LIN {X 0,Y 466.737,Z 357.71,A -85,B 0,C 180,E1 -7511.495,E2 -7511.495} C_VEL
LIN {X 0,Y 466.868,Z 355.189,A -85,B 0,C 180,E1 -7512.642,E2 -7512.642} C_VEL
LIN {X 0,Y 467.016,Z 350.85,A -85,B 0,C 180,E1 -7514.108,E2 -7514.108} C_VEL
LIN {X 0,Y 467.238,Z 344.895,A -85,B 0,C 180,E1 -7515.6,E2 -7515.6} C_VEL
LIN {X 0,Y 467.572,Z 338.558,A -85,B 0,C 180,E1 -7516.852,E2 -7516.852} C_VEL
LIN {X 0,Y 468.005,Z 329.992,A -85,B 0,C 180,E1 -7518.213,E2 -7518.213} C_VEL
LIN {X 0,Y 468.461,Z 320.576,A -85,B 0,C 180,E1 -7519.404,E2 -7519.404} C_VEL
LIN {X 0,Y 468.938,Z 310.487,A -85,B 0,C 180,E1 -7520.436,E2 -7520.436} C_VEL
LIN {X 0,Y 469.406,Z 299.87,A -85,B 0,C 180,E1 -7521.312,E2 -7521.312} C_VEL
LIN {X 0,Y 469.889,Z 288.638,A -85,B 0,C 180,E1 -7522.042,E2 -7522.042} C_VEL
LIN {X 0,Y 470.257,Z 275.513,A -85,B 0,C 180,E1 -7522.685,E2 -7522.685} C_VEL
LIN {X 0,Y 470.519,Z 262.558,A -85,B 0,C 180,E1 -7523.128,E2 -7523.128} C_VEL
LIN {X 0,Y 470.697,Z 246.728,A -85,B 0,C 180,E1 -7523.438,E2 -7523.438} C_VEL
LIN {X 0,Y 471.435,Z 164.016,A -85,B 0,C 180,E1 -7524.746,E2 -7524.746} C_VEL
LIN {X 0,Y 468.633,Z 150.697,A -85,B 0,C 180,E1 -7525.095,E2 -7525.095} C_VEL
LIN {X 0,Y 468.758,Z 142.318,A -85,B 0,C 180,E1 -7526.795,E2 -7526.795} C_VEL
LIN {X 0,Y 467.609,Z 135.273,A -85,B 0,C 180,E1 -7528.289,E2 -7528.289} C_VEL
LIN {X 0,Y 467.577,Z 135.244,A -85,B 0,C 180,E1 -7531.251,E2 -7531.251} C_VEL
LIN {X 0,Y 467.591,Z 135.241,A -85,B 0,C 180,E1 -7534.159,E2 -7534.159} C_VEL
LIN {X 0,Y 467.579,Z 135.247,A -85,B 0,C 180,E1 -7536.997,E2 -7536.997} C_VEL
LIN {X 0,Y 467.625,Z 135.234,A -85,B 0,C 180,E1 -7539.778,E2 -7539.778} C_VEL
LIN {X 0,Y 467.598,Z 135.239,A -85,B 0,C 180,E1 -7542.507,E2 -7542.507} C_VEL
LIN {X 0,Y 467.606,Z 135.24,A -85,B 0,C 180,E1 -7545.197,E2 -7545.197} C_VEL
LIN {X 0,Y 467.66,Z 135.231,A -85,B 0,C 180,E1 -7547.855,E2 -7547.855} C_VEL
LIN {X 0,Y 467.671,Z 135.229,A -85,B 0,C 180,E1 -7551.358,E2 -7551.358} C_VEL
LIN {X 0,Y 467.709,Z 135.225,A -85,B 0,C 180,E1 -7553.963,E2 -7553.963} C_VEL
LIN {X 0,Y 467.818,Z 135.209,A -85,B 0,C 180,E1 -7557.417,E2 -7557.417} C_VEL
LIN {X 0,Y 467.854,Z 135.204,A -85,B 0,C 180,E1 -7560,E2 -7560} C_VEL
LIN {X 0,Y 467.816,Z 135.207,A -85,B 0,C 180,E1 -7562.584,E2 -7562.584} C_VEL
LIN {X 0,Y 467.705,Z 135.225,A -85,B 0,C 180,E1 -7566.038,E2 -7566.038} C_VEL
LIN {X 0,Y 467.634,Z 135.231,A -85,B 0,C 180,E1 -7568.644,E2 -7568.644} C_VEL
LIN {X 0,Y 467.646,Z 135.232,A -85,B 0,C 180,E1 -7572.146,E2 -7572.146} C_VEL
LIN {X 0,Y 467.581,Z 135.239,A -85,B 0,C 180,E1 -7575.697,E2 -7575.697} C_VEL
LIN {X 0,Y 467.553,Z 135.239,A -85,B 0,C 180,E1 -7578.739,E2 -7578.739} C_VEL
LIN {X 0,Y 467.52,Z 135.246,A -85,B 0,C 180,E1 -7582.075,E2 -7582.075} C_VEL
LIN {X 0,Y 467.533,Z 135.244,A -85,B 0,C 180,E1 -7584.892,E2 -7584.892} C_VEL
LIN {X 0,Y 467.542,Z 135.241,A -85,B 0,C 180,E1 -7587.775,E2 -7587.775} C_VEL
LIN {X 0,Y 467.534,Z 135.247,A -85,B 0,C 180,E1 -7591.037,E2 -7591.037} C_VEL
LIN {X 0,Y 467.571,Z 135.239,A -85,B 0,C 180,E1 -7593.79,E2 -7593.79} C_VEL
LIN {X 0,Y 467.529,Z 135.25,A -85,B 0,C 180,E1 -7596.963,E2 -7596.963} C_VEL
LIN {X 0,Y 467.568,Z 135.24,A -85,B 0,C 180,E1 -7599.951,E2 -7599.951} C_VEL
LIN {X 0,Y 467.524,Z 135.251,A -85,B 0,C 180,E1 -7602.568,E2 -7602.568} C_VEL
LIN {X 0,Y 467.57,Z 135.244,A -85,B 0,C 180,E1 -7605.052,E2 -7605.052} C_VEL
LIN {X 0,Y 467.571,Z 135.245,A -85,B 0,C 180,E1 -7608.725,E2 -7608.725} C_VEL
LIN {X 0,Y 467.566,Z 135.244,A -85,B 0,C 180,E1 -7611.955,E2 -7611.955} C_VEL
LIN {X 0,Y 467.567,Z 135.241,A -85,B 0,C 180,E1 -7615.167,E2 -7615.167} C_VEL
LIN {X 0,Y 467.587,Z 135.247,A -85,B 0,C 180,E1 -7618.26,E2 -7618.26} C_VEL
LIN {X 0,Y 467.56,Z 135.243,A -85,B 0,C 180,E1 -7621.249,E2 -7621.249} C_VEL
LIN {X 0,Y 467.611,Z 135.331,A -85,B 0,C 180,E1 -7623.65,E2 -7623.65} C_VEL
LIN {X 0,Y 469.706,Z 145.922,A -85,B 0,C 180,E1 -7625.6,E2 -7625.6} C_VEL
LIN {X 0,Y 469.617,Z 153.321,A -85,B 0,C 180,E1 -7626.868,E2 -7626.868} C_VEL
LIN {X 0,Y 468.886,Z 169.647,A -85,B 0,C 180,E1 -7629.605,E2 -7629.605} C_VEL
LIN {X 0,Y 468.398,Z 184.571,A -85,B 0,C 180,E1 -7632.085,E2 -7632.085} C_VEL
LIN {X 0,Y 468.222,Z 189.663,A -85,B 0,C 180,E1 -7632.927,E2 -7632.927} C_VEL
LIN {X 0,Y 471.192,Z 210.245,A -85,B 0,C 180,E1 -7633.383,E2 -7633.383} C_VEL
LIN {X 0,Y 470.478,Z 298.444,A -85,B 0,C 180,E1 -7634.79,E2 -7634.79} C_VEL
LIN {X 0,Y 470.078,Z 311.692,A -85,B 0,C 180,E1 -7635.165,E2 -7635.165} C_VEL
LIN {X 0,Y 469.572,Z 324.447,A -85,B 0,C 180,E1 -7635.702,E2 -7635.702} C_VEL
LIN {X 0,Y 469.102,Z 335.815,A -85,B 0,C 180,E1 -7636.351,E2 -7636.351} C_VEL
LIN {X 0,Y 468.602,Z 347.595,A -85,B 0,C 180,E1 -7637.222,E2 -7637.222} C_VEL
LIN {X 0,Y 468.114,Z 358.121,A -85,B 0,C 180,E1 -7638.196,E2 -7638.196} C_VEL
LIN {X 0,Y 467.705,Z 366.768,A -85,B 0,C 180,E1 -7639.173,E2 -7639.173} C_VEL
LIN {X 0,Y 467.358,Z 374.752,A -85,B 0,C 180,E1 -7640.26,E2 -7640.26} C_VEL
LIN {X 0,Y 467.021,Z 382.558,A -85,B 0,C 180,E1 -7641.562,E2 -7641.562} C_VEL
LIN {X 0,Y 466.83,Z 389.753,A -85,B 0,C 180,E1 -7643.082,E2 -7643.082} C_VEL
LIN {X 0,Y 466.724,Z 394.545,A -85,B 0,C 180,E1 -7644.383,E2 -7644.383} C_VEL
LIN {X 0,Y 466.648,Z 398.21,A -85,B 0,C 180,E1 -7645.681,E2 -7645.681} C_VEL
LIN {X 0,Y 466.701,Z 400.106,A -85,B 0,C 180,E1 -7646.546,E2 -7646.546} C_VEL
LIN {X 0,Y 466.685,Z 401.527,A -85,B 0,C 180,E1 -7647.41,E2 -7647.41} C_VEL
LIN {X 0,Y 466.663,Z 402.544,A -85,B 0,C 180,E1 -7648.273,E2 -7648.273} C_VEL
LIN {X 0,Y 466.627,Z 403.166,A -85,B 0,C 180,E1 -7649.137,E2 -7649.137} C_VEL
LIN {X 0,Y 466.611,Z 403.39,A -85,B 0,C 180,E1 -7650,E2 -7650} C_VEL
LIN {X 0,Y 466.627,Z 403.176,A -85,B 0,C 180,E1 -7650.862,E2 -7650.862} C_VEL
LIN {X 0,Y 466.662,Z 402.569,A -85,B 0,C 180,E1 -7651.726,E2 -7651.726} C_VEL
LIN {X 0,Y 466.685,Z 401.567,A -85,B 0,C 180,E1 -7652.589,E2 -7652.589} C_VEL
LIN {X 0,Y 466.7,Z 400.153,A -85,B 0,C 180,E1 -7653.453,E2 -7653.453} C_VEL
LIN {X 0,Y 466.687,Z 397.184,A -85,B 0,C 180,E1 -7654.751,E2 -7654.751} C_VEL
LIN {X 0,Y 466.73,Z 393.159,A -85,B 0,C 180,E1 -7656.05,E2 -7656.05} C_VEL
LIN {X 0,Y 466.905,Z 386.961,A -85,B 0,C 180,E1 -7657.568,E2 -7657.568} C_VEL
LIN {X 0,Y 467.11,Z 380.195,A -85,B 0,C 180,E1 -7658.871,E2 -7658.871} C_VEL
LIN {X 0,Y 467.436,Z 371.798,A -85,B 0,C 180,E1 -7660.175,E2 -7660.175} C_VEL
LIN {X 0,Y 467.88,Z 363.155,A -85,B 0,C 180,E1 -7661.26,E2 -7661.26} C_VEL
LIN {X 0,Y 468.334,Z 353.176,A -85,B 0,C 180,E1 -7662.284,E2 -7662.284} C_VEL
LIN {X 0,Y 468.807,Z 341.931,A -85,B 0,C 180,E1 -7663.215,E2 -7663.215} C_VEL
LIN {X 0,Y 469.324,Z 330.244,A -85,B 0,C 180,E1 -7663.973,E2 -7663.973} C_VEL
LIN {X 0,Y 469.784,Z 318.114,A -85,B 0,C 180,E1 -7664.567,E2 -7664.567} C_VEL
LIN {X 0,Y 470.223,Z 304.953,A -85,B 0,C 180,E1 -7665.023,E2 -7665.023} C_VEL
LIN {X 0,Y 470.436,Z 292.277,A -85,B 0,C 180,E1 -7665.294,E2 -7665.294} C_VEL
LIN {X 0,Y 471.011,Z 209.547,A -85,B 0,C 180,E1 -7666.591,E2 -7666.591} C_VEL
LIN {X 0,Y 468.278,Z 190.339,A -85,B 0,C 180,E1 -7667.017,E2 -7667.017} C_VEL
LIN {X 0,Y 468.949,Z 171.549,A -85,B 0,C 180,E1 -7670.163,E2 -7670.163} C_VEL
LIN {X 0,Y 469.833,Z 152.715,A -85,B 0,C 180,E1 -7673.353,E2 -7673.353} C_VEL
LIN {X 0,Y 469.889,Z 146.56,A -85,B 0,C 180,E1 -7674.418,E2 -7674.418} C_VEL
LIN {X 0,Y 467.649,Z 135.235,A -85,B 0,C 180,E1 -7676.557,E2 -7676.557} C_VEL
LIN {X 0,Y 467.554,Z 135.246,A -85,B 0,C 180,E1 -7679.738,E2 -7679.738} C_VEL
LIN {X 0,Y 467.584,Z 135.237,A -85,B 0,C 180,E1 -7682.758,E2 -7682.758} C_VEL
LIN {X 0,Y 467.554,Z 135.247,A -85,B 0,C 180,E1 -7685.889,E2 -7685.889} C_VEL
LIN {X 0,Y 467.583,Z 135.237,A -85,B 0,C 180,E1 -7689.144,E2 -7689.144} C_VEL
LIN {X 0,Y 467.587,Z 135.236,A -85,B 0,C 180,E1 -7692.566,E2 -7692.566} C_VEL
LIN {X 0,Y 467.566,Z 135.239,A -85,B 0,C 180,E1 -7695.052,E2 -7695.052} C_VEL
LIN {X 0,Y 467.589,Z 135.24,A -85,B 0,C 180,E1 -7697.439,E2 -7697.439} C_VEL
LIN {X 0,Y 467.56,Z 135.239,A -85,B 0,C 180,E1 -7700.853,E2 -7700.853} C_VEL
LIN {X 0,Y 467.558,Z 135.24,A -85,B 0,C 180,E1 -7704.261,E2 -7704.261} C_VEL
LIN {X 0,Y 467.578,Z 135.242,A -85,B 0,C 180,E1 -7707.321,E2 -7707.321} C_VEL
LIN {X 0,Y 467.568,Z 135.238,A -85,B 0,C 180,E1 -7710.667,E2 -7710.667} C_VEL
LIN {X 0,Y 467.616,Z 135.238,A -85,B 0,C 180,E1 -7713.199,E2 -7713.199} C_VEL
LIN {X 0,Y 467.591,Z 135.235,A -85,B 0,C 180,E1 -7716.468,E2 -7716.468} C_VEL
LIN {X 0,Y 467.621,Z 135.233,A -85,B 0,C 180,E1 -7719.777,E2 -7719.777} C_VEL
LIN {X 0,Y 467.597,Z 135.235,A -85,B 0,C 180,E1 -7722.506,E2 -7722.506} C_VEL
LIN {X 0,Y 467.606,Z 135.241,A -85,B 0,C 180,E1 -7725.196,E2 -7725.196} C_VEL
LIN {X 0,Y 467.655,Z 135.228,A -85,B 0,C 180,E1 -7727.854,E2 -7727.854} C_VEL
LIN {X 0,Y 467.68,Z 135.228,A -85,B 0,C 180,E1 -7731.357,E2 -7731.357} C_VEL
LIN {X 0,Y 467.734,Z 135.217,A -85,B 0,C 180,E1 -7733.962,E2 -7733.962} C_VEL
LIN {X 0,Y 467.858,Z 135.204,A -85,B 0,C 180,E1 -7737.417,E2 -7737.417} C_VEL
LIN {X 0,Y 467.881,Z 135.199,A -85,B 0,C 180,E1 -7740,E2 -7740} C_VEL
LIN {X 0,Y 467.858,Z 135.207,A -85,B 0,C 180,E1 -7742.582,E2 -7742.582} C_VEL
LIN {X 0,Y 467.734,Z 135.218,A -85,B 0,C 180,E1 -7746.037,E2 -7746.037} C_VEL
LIN {X 0,Y 467.679,Z 135.232,A -85,B 0,C 180,E1 -7748.642,E2 -7748.642} C_VEL
LIN {X 0,Y 467.653,Z 135.23,A -85,B 0,C 180,E1 -7752.145,E2 -7752.145} C_VEL
LIN {X 0,Y 467.636,Z 135.23,A -85,B 0,C 180,E1 -7755.695,E2 -7755.695} C_VEL
LIN {X 0,Y 467.614,Z 135.236,A -85,B 0,C 180,E1 -7758.764,E2 -7758.764} C_VEL
LIN {X 0,Y 467.577,Z 135.237,A -85,B 0,C 180,E1 -7761.268,E2 -7761.268} C_VEL
LIN {X 0,Y 467.568,Z 135.241,A -85,B 0,C 180,E1 -7763.943,E2 -7763.943} C_VEL
LIN {X 0,Y 467.624,Z 135.233,A -85,B 0,C 180,E1 -7766.799,E2 -7766.799} C_VEL
LIN {X 0,Y 467.55,Z 135.242,A -85,B 0,C 180,E1 -7769.738,E2 -7769.738} C_VEL
LIN {X 0,Y 467.579,Z 135.238,A -85,B 0,C 180,E1 -7772.758,E2 -7772.758} C_VEL
LIN {X 0,Y 467.552,Z 135.245,A -85,B 0,C 180,E1 -7775.889,E2 -7775.889} C_VEL
LIN {X 0,Y 467.614,Z 135.232,A -85,B 0,C 180,E1 -7779.141,E2 -7779.141} C_VEL
LIN {X 0,Y 467.614,Z 135.234,A -85,B 0,C 180,E1 -7782.571,E2 -7782.571} C_VEL
LIN {X 0,Y 467.569,Z 135.242,A -85,B 0,C 180,E1 -7786.176,E2 -7786.176} C_VEL
LIN {X 0,Y 467.585,Z 135.236,A -85,B 0,C 180,E1 -7788.721,E2 -7788.721} C_VEL
LIN {X 0,Y 467.573,Z 135.241,A -85,B 0,C 180,E1 -7791.407,E2 -7791.407} C_VEL
LIN {X 0,Y 467.557,Z 135.241,A -85,B 0,C 180,E1 -7794.26,E2 -7794.26} C_VEL
LIN {X 0,Y 467.577,Z 135.241,A -85,B 0,C 180,E1 -7797.321,E2 -7797.321} C_VEL
LIN {X 0,Y 467.565,Z 135.238,A -85,B 0,C 180,E1 -7800.667,E2 -7800.667} C_VEL
LIN {X 0,Y 467.623,Z 135.235,A -85,B 0,C 180,E1 -7803.201,E2 -7803.201} C_VEL
LIN {X 0,Y 467.588,Z 135.236,A -85,B 0,C 180,E1 -7806.468,E2 -7806.468} C_VEL
LIN {X 0,Y 467.619,Z 135.235,A -85,B 0,C 180,E1 -7809.778,E2 -7809.778} C_VEL
LIN {X 0,Y 467.604,Z 135.234,A -85,B 0,C 180,E1 -7812.507,E2 -7812.507} C_VEL
LIN {X 0,Y 467.596,Z 135.238,A -85,B 0,C 180,E1 -7815.421,E2 -7815.421} C_VEL
LIN {X 0,Y 466.925,Z 135.32,A -85,B 0,C 180,E1 -7816.14,E2 -7816.14} C_VEL
LIN {X 0,Y 464.08,Z 135.68,A -85,B 0,C 180,E1 -7817.309,E2 -7817.309} C_VEL
LIN {X 0,Y 461.681,Z 135.974,A -85,B 0,C 180,E1 -7818.251,E2 -7818.251} C_VEL
LIN {X 0,Y 460.656,Z 136.104,A -85,B 0,C 180,E1 -7818.978,E2 -7818.978} C_VEL
LIN {X 0,Y 460.574,Z 136.112,A -85,B 0,C 180,E1 -7819.225,E2 -7819.225} C_VEL
LIN {X 0,Y 460.716,Z 136.093,A -85,B 0,C 180,E1 -7822.538,E2 -7822.538} C_VEL
LIN {X 0,Y 460.696,Z 136.098,A -85,B 0,C 180,E1 -7824.749,E2 -7824.749} C_VEL
LIN {X 0,Y 460.822,Z 136.082,A -85,B 0,C 180,E1 -7827.378,E2 -7827.378} C_VEL
LIN {X 0,Y 460.85,Z 136.075,A -85,B 0,C 180,E1 -7830.001,E2 -7830.001} C_VEL
LIN {X 0,Y 460.822,Z 136.082,A -85,B 0,C 180,E1 -7832.623,E2 -7832.623} C_VEL
LIN {X 0,Y 460.709,Z 136.093,A -85,B 0,C 180,E1 -7836.13,E2 -7836.13} C_VEL
LIN {X 0,Y 460.626,Z 136.111,A -85,B 0,C 180,E1 -7838.777,E2 -7838.777} C_VEL
LIN {X 0,Y 460.611,Z 136.109,A -85,B 0,C 180,E1 -7842.446,E2 -7842.446} C_VEL
LIN {X 0,Y 460.581,Z 136.113,A -85,B 0,C 180,E1 -7845.991,E2 -7845.991} C_VEL
LIN {X 0,Y 460.632,Z 136.132,A -85,B 0,C 180,E1 -7847.71,E2 -7847.71} C_VEL
LIN {X 0,Y 461.679,Z 143.329,A -85,B 0,C 180,E1 -7849.301,E2 -7849.301} C_VEL
LIN {X 0,Y 461.56,Z 150.531,A -85,B 0,C 180,E1 -7850.821,E2 -7850.821} C_VEL
LIN {X 0,Y 464.547,Z 166.407,A -85,B 0,C 180,E1 -7851.203,E2 -7851.203} C_VEL
LIN {X 0,Y 463.605,Z 257.763,A -85,B 0,C 180,E1 -7852.675,E2 -7852.675} C_VEL
LIN {X 0,Y 463.304,Z 271.247,A -85,B 0,C 180,E1 -7853.074,E2 -7853.074} C_VEL
LIN {X 0,Y 463.029,Z 283.235,A -85,B 0,C 180,E1 -7853.599,E2 -7853.599} C_VEL
LIN {X 0,Y 462.661,Z 295.098,A -85,B 0,C 180,E1 -7854.299,E2 -7854.299} C_VEL
LIN {X 0,Y 462.054,Z 307.015,A -85,B 0,C 180,E1 -7855.208,E2 -7855.208} C_VEL
LIN {X 0,Y 461.572,Z 317.396,A -85,B 0,C 180,E1 -7856.204,E2 -7856.204} C_VEL
LIN {X 0,Y 461.141,Z 325.924,A -85,B 0,C 180,E1 -7857.208,E2 -7857.208} C_VEL
LIN {X 0,Y 460.718,Z 334.657,A -85,B 0,C 180,E1 -7858.471,E2 -7858.471} C_VEL
LIN {X 0,Y 460.34,Z 342.39,A -85,B 0,C 180,E1 -7859.86,E2 -7859.86} C_VEL
LIN {X 0,Y 460.026,Z 348.699,A -85,B 0,C 180,E1 -7861.295,E2 -7861.295} C_VEL
LIN {X 0,Y 459.811,Z 353.709,A -85,B 0,C 180,E1 -7862.792,E2 -7862.792} C_VEL
LIN {X 0,Y 459.632,Z 357.471,A -85,B 0,C 180,E1 -7864.343,E2 -7864.343} C_VEL
LIN {X 0,Y 459.521,Z 359.841,A -85,B 0,C 180,E1 -7865.847,E2 -7865.847} C_VEL
LIN {X 0,Y 459.475,Z 360.994,A -85,B 0,C 180,E1 -7867.31,E2 -7867.31} C_VEL
LIN {X 0,Y 459.466,Z 361.006,A -85,B 0,C 180,E1 -7868.84,E2 -7868.84} C_VEL
LIN {X 0,Y 459.514,Z 360.091,A -85,B 0,C 180,E1 -7870.119,E2 -7870.119} C_VEL
LIN {X 0,Y 459.662,Z 358.162,A -85,B 0,C 180,E1 -7871.481,E2 -7871.481} C_VEL
LIN {X 0,Y 459.802,Z 355.31,A -85,B 0,C 180,E1 -7872.806,E2 -7872.806} C_VEL
LIN {X 0,Y 459.947,Z 351.531,A -85,B 0,C 180,E1 -7874.098,E2 -7874.098} C_VEL
LIN {X 0,Y 460.193,Z 345.858,A -85,B 0,C 180,E1 -7875.582,E2 -7875.582} C_VEL
LIN {X 0,Y 460.525,Z 339.461,A -85,B 0,C 180,E1 -7876.889,E2 -7876.889} C_VEL
LIN {X 0,Y 460.936,Z 331.969,A -85,B 0,C 180,E1 -7878.128,E2 -7878.128} C_VEL
LIN {X 0,Y 461.43,Z 322.724,A -85,B 0,C 180,E1 -7879.37,E2 -7879.37} C_VEL
LIN {X 0,Y 461.963,Z 312.724,A -85,B 0,C 180,E1 -7880.449,E2 -7880.449} C_VEL
LIN {X 0,Y 462.4,Z 302.857,A -85,B 0,C 180,E1 -7881.313,E2 -7881.313} C_VEL
LIN {X 0,Y 462.968,Z 291.132,A -85,B 0,C 180,E1 -7882.128,E2 -7882.128} C_VEL
LIN {X 0,Y 463.389,Z 279.131,A -85,B 0,C 180,E1 -7882.769,E2 -7882.769} C_VEL
LIN {X 0,Y 463.589,Z 266.908,A -85,B 0,C 180,E1 -7883.242,E2 -7883.242} C_VEL
LIN {X 0,Y 463.87,Z 253.753,A -85,B 0,C 180,E1 -7883.564,E2 -7883.564} C_VEL
LIN {X 0,Y 464.616,Z 164.695,A -85,B 0,C 180,E1 -7885.004,E2 -7885.004} C_VEL
LIN {X 0,Y 461.721,Z 151.061,A -85,B 0,C 180,E1 -7885.36,E2 -7885.36} C_VEL
LIN {X 0,Y 461.749,Z 142.764,A -85,B 0,C 180,E1 -7887.066,E2 -7887.066} C_VEL
LIN {X 0,Y 460.537,Z 136.122,A -85,B 0,C 180,E1 -7888.515,E2 -7888.515} C_VEL
LIN {X 0,Y 460.552,Z 136.119,A -85,B 0,C 180,E1 -7891.768,E2 -7891.768} C_VEL
LIN {X 0,Y 460.536,Z 136.122,A -85,B 0,C 180,E1 -7894.705,E2 -7894.705} C_VEL
LIN {X 0,Y 460.513,Z 136.123,A -85,B 0,C 180,E1 -7897.572,E2 -7897.572} C_VEL
LIN {X 0,Y 460.571,Z 136.114,A -85,B 0,C 180,E1 -7900.385,E2 -7900.385} C_VEL
LIN {X 0,Y 460.608,Z 136.108,A -85,B 0,C 180,E1 -7904.06,E2 -7904.06} C_VEL
LIN {X 0,Y 460.614,Z 136.108,A -85,B 0,C 180,E1 -7907.666,E2 -7907.666} C_VEL
LIN {X 0,Y 460.622,Z 136.108,A -85,B 0,C 180,E1 -7911.224,E2 -7911.224} C_VEL
LIN {X 0,Y 460.675,Z 136.101,A -85,B 0,C 180,E1 -7913.87,E2 -7913.87} C_VEL
LIN {X 0,Y 460.762,Z 136.088,A -85,B 0,C 180,E1 -7917.378,E2 -7917.378} C_VEL
LIN {X 0,Y 460.823,Z 136.08,A -85,B 0,C 180,E1 -7920,E2 -7920} C_VEL
LIN {X 0,Y 460.76,Z 136.085,A -85,B 0,C 180,E1 -7922.623,E2 -7922.623} C_VEL
LIN {X 0,Y 460.671,Z 136.099,A -85,B 0,C 180,E1 -7926.131,E2 -7926.131} C_VEL
LIN {X 0,Y 460.589,Z 136.108,A -85,B 0,C 180,E1 -7928.777,E2 -7928.777} C_VEL
LIN {X 0,Y 460.602,Z 136.107,A -85,B 0,C 180,E1 -7932.435,E2 -7932.435} C_VEL
LIN {X 0,Y 460.531,Z 136.119,A -85,B 0,C 180,E1 -7935.965,E2 -7935.965} C_VEL
LIN {X 0,Y 460.514,Z 136.117,A -85,B 0,C 180,E1 -7938.879,E2 -7938.879} C_VEL
LIN {X 0,Y 460.494,Z 136.12,A -85,B 0,C 180,E1 -7942.43,E2 -7942.43} C_VEL
LIN {X 0,Y 460.526,Z 136.119,A -85,B 0,C 180,E1 -7945.79,E2 -7945.79} C_VEL
LIN {X 0,Y 460.5,Z 136.117,A -85,B 0,C 180,E1 -7948.237,E2 -7948.237} C_VEL
LIN {X 0,Y 460.5,Z 136.121,A -85,B 0,C 180,E1 -7951.277,E2 -7951.277} C_VEL
LIN {X 0,Y 460.527,Z 136.118,A -85,B 0,C 180,E1 -7954.503,E2 -7954.503} C_VEL
LIN {X 0,Y 460.503,Z 136.119,A -85,B 0,C 180,E1 -7957.623,E2 -7957.623} C_VEL
LIN {X 0,Y 460.519,Z 136.12,A -85,B 0,C 180,E1 -7961.013,E2 -7961.013} C_VEL
LIN {X 0,Y 460.516,Z 136.124,A -85,B 0,C 180,E1 -7964.589,E2 -7964.589} C_VEL
LIN {X 0,Y 460.496,Z 136.124,A -85,B 0,C 180,E1 -7967.815,E2 -7967.815} C_VEL
LIN {X 0,Y 460.519,Z 136.124,A -85,B 0,C 180,E1 -7970.136,E2 -7970.136} C_VEL
LIN {X 0,Y 460.477,Z 136.124,A -85,B 0,C 180,E1 -7973.47,E2 -7973.47} C_VEL
LIN {X 0,Y 460.534,Z 136.123,A -85,B 0,C 180,E1 -7976.675,E2 -7976.675} C_VEL
LIN {X 0,Y 460.512,Z 136.125,A -85,B 0,C 180,E1 -7979.759,E2 -7979.759} C_VEL
LIN {X 0,Y 460.544,Z 136.119,A -85,B 0,C 180,E1 -7982.754,E2 -7982.754} C_VEL
LIN {X 0,Y 460.598,Z 136.268,A -85,B 0,C 180,E1 -7983.431,E2 -7983.431} C_VEL
LIN {X 0,Y 462.885,Z 148.084,A -85,B 0,C 180,E1 -7985.642,E2 -7985.642} C_VEL
LIN {X 0,Y 462.385,Z 161.772,A -85,B 0,C 180,E1 -7987.998,E2 -7987.998} C_VEL
LIN {X 0,Y 461.576,Z 181.577,A -85,B 0,C 180,E1 -7991.352,E2 -7991.352} C_VEL
LIN {X 0,Y 461.259,Z 189.355,A -85,B 0,C 180,E1 -7992.657,E2 -7992.657} C_VEL
LIN {X 0,Y 464.392,Z 210.611,A -85,B 0,C 180,E1 -7993.135,E2 -7993.135} C_VEL
LIN {X 0,Y 463.632,Z 298.318,A -85,B 0,C 180,E1 -7994.56,E2 -7994.56} C_VEL
LIN {X 0,Y 463.22,Z 311.48,A -85,B 0,C 180,E1 -7994.94,E2 -7994.94} C_VEL
LIN {X 0,Y 462.696,Z 324.192,A -85,B 0,C 180,E1 -7995.485,E2 -7995.485} C_VEL
LIN {X 0,Y 462.189,Z 335.53,A -85,B 0,C 180,E1 -7996.143,E2 -7996.143} C_VEL
LIN {X 0,Y 461.694,Z 346.551,A -85,B 0,C 180,E1 -7996.964,E2 -7996.964} C_VEL
LIN {X 0,Y 461.109,Z 357.818,A -85,B 0,C 180,E1 -7998.014,E2 -7998.014} C_VEL
LIN {X 0,Y 460.717,Z 366.463,A -85,B 0,C 180,E1 -7999.007,E2 -7999.007} C_VEL
LIN {X 0,Y 460.301,Z 374.441,A -85,B 0,C 180,E1 -8000.109,E2 -8000.109} C_VEL
LIN {X 0,Y 459.969,Z 382.243,A -85,B 0,C 180,E1 -8001.432,E2 -8001.432} C_VEL
LIN {X 0,Y 459.742,Z 389.434,A -85,B 0,C 180,E1 -8002.975,E2 -8002.975} C_VEL
LIN {X 0,Y 459.624,Z 394.225,A -85,B 0,C 180,E1 -8004.295,E2 -8004.295} C_VEL
LIN {X 0,Y 459.565,Z 397.891,A -85,B 0,C 180,E1 -8005.614,E2 -8005.614} C_VEL
LIN {X 0,Y 459.597,Z 399.785,A -85,B 0,C 180,E1 -8006.493,E2 -8006.493} C_VEL
LIN {X 0,Y 459.606,Z 401.207,A -85,B 0,C 180,E1 -8007.37,E2 -8007.37} C_VEL
LIN {X 0,Y 459.56,Z 402.846,A -85,B 0,C 180,E1 -8009.123,E2 -8009.123} C_VEL
LIN {X 0,Y 459.542,Z 403.067,A -85,B 0,C 180,E1 -8009.999,E2 -8009.999} C_VEL
LIN {X 0,Y 459.56,Z 402.85,A -85,B 0,C 180,E1 -8010.876,E2 -8010.876} C_VEL
LIN {X 0,Y 459.605,Z 401.237,A -85,B 0,C 180,E1 -8012.629,E2 -8012.629} C_VEL
LIN {X 0,Y 459.597,Z 399.817,A -85,B 0,C 180,E1 -8013.506,E2 -8013.506} C_VEL
LIN {X 0,Y 459.614,Z 396.843,A -85,B 0,C 180,E1 -8014.824,E2 -8014.824} C_VEL
LIN {X 0,Y 459.675,Z 391.923,A -85,B 0,C 180,E1 -8016.386,E2 -8016.386} C_VEL
LIN {X 0,Y 459.867,Z 385.582,A -85,B 0,C 180,E1 -8017.905,E2 -8017.905} C_VEL
LIN {X 0,Y 460.147,Z 378.574,A -85,B 0,C 180,E1 -8019.228,E2 -8019.228} C_VEL
LIN {X 0,Y 460.496,Z 369.778,A -85,B 0,C 180,E1 -8020.552,E2 -8020.552} C_VEL
LIN {X 0,Y 461.056,Z 359.794,A -85,B 0,C 180,E1 -8021.763,E2 -8021.763} C_VEL
LIN {X 0,Y 461.506,Z 349.411,A -85,B 0,C 180,E1 -8022.776,E2 -8022.776} C_VEL
LIN {X 0,Y 462.054,Z 338.372,A -85,B 0,C 180,E1 -8023.636,E2 -8023.636} C_VEL
LIN {X 0,Y 462.506,Z 327.719,A -85,B 0,C 180,E1 -8024.295,E2 -8024.295} C_VEL
LIN {X 0,Y 462.991,Z 316.217,A -85,B 0,C 180,E1 -8024.842,E2 -8024.842} C_VEL
LIN {X 0,Y 463.347,Z 304.236,A -85,B 0,C 180,E1 -8025.252,E2 -8025.252} C_VEL
LIN {X 0,Y 463.626,Z 289.449,A -85,B 0,C 180,E1 -8025.552,E2 -8025.552} C_VEL
LIN {X 0,Y 464.141,Z 209.997,A -85,B 0,C 180,E1 -8026.822,E2 -8026.822} C_VEL
LIN {X 0,Y 461.259,Z 190.058,A -85,B 0,C 180,E1 -8027.271,E2 -8027.271} C_VEL
LIN {X 0,Y 461.978,Z 172.539,A -85,B 0,C 180,E1 -8030.248,E2 -8030.248} C_VEL
LIN {X 0,Y 462.957,Z 152.355,A -85,B 0,C 180,E1 -8033.721,E2 -8033.721} C_VEL
LIN {X 0,Y 463.026,Z 148.507,A -85,B 0,C 180,E1 -8034.396,E2 -8034.396} C_VEL
LIN {X 0,Y 460.603,Z 136.113,A -85,B 0,C 180,E1 -8036.751,E2 -8036.751} C_VEL
LIN {X 0,Y 460.511,Z 136.124,A -85,B 0,C 180,E1 -8040.239,E2 -8040.239} C_VEL
LIN {X 0,Y 460.53,Z 136.116,A -85,B 0,C 180,E1 -8043.324,E2 -8043.324} C_VEL
LIN {X 0,Y 460.477,Z 136.123,A -85,B 0,C 180,E1 -8046.529,E2 -8046.529} C_VEL
LIN {X 0,Y 460.558,Z 136.12,A -85,B 0,C 180,E1 -8049.859,E2 -8049.859} C_VEL
LIN {X 0,Y 460.512,Z 136.117,A -85,B 0,C 180,E1 -8052.9,E2 -8052.9} C_VEL
LIN {X 0,Y 460.509,Z 136.125,A -85,B 0,C 180,E1 -8055.83,E2 -8055.83} C_VEL
LIN {X 0,Y 460.53,Z 136.116,A -85,B 0,C 180,E1 -8058.988,E2 -8058.988} C_VEL
LIN {X 0,Y 460.518,Z 136.12,A -85,B 0,C 180,E1 -8061.266,E2 -8061.266} C_VEL
LIN {X 0,Y 460.507,Z 136.118,A -85,B 0,C 180,E1 -8064.554,E2 -8064.554} C_VEL
LIN {X 0,Y 460.529,Z 136.12,A -85,B 0,C 180,E1 -8067.715,E2 -8067.715} C_VEL
LIN {X 0,Y 460.538,Z 136.115,A -85,B 0,C 180,E1 -8070.768,E2 -8070.768} C_VEL
LIN {X 0,Y 460.562,Z 136.114,A -85,B 0,C 180,E1 -8073.734,E2 -8073.734} C_VEL
LIN {X 0,Y 460.545,Z 136.114,A -85,B 0,C 180,E1 -8076.623,E2 -8076.623} C_VEL
LIN {X 0,Y 460.55,Z 136.118,A -85,B 0,C 180,E1 -8079.452,E2 -8079.452} C_VEL
LIN {X 0,Y 460.548,Z 136.113,A -85,B 0,C 180,E1 -8082.229,E2 -8082.229} C_VEL
LIN {X 0,Y 460.564,Z 136.116,A -85,B 0,C 180,E1 -8084.964,E2 -8084.964} C_VEL
LIN {X 0,Y 460.61,Z 136.107,A -85,B 0,C 180,E1 -8088.559,E2 -8088.559} C_VEL
LIN {X 0,Y 460.694,Z 136.095,A -85,B 0,C 180,E1 -8092.108,E2 -8092.108} C_VEL
LIN {X 0,Y 460.693,Z 136.1,A -85,B 0,C 180,E1 -8094.748,E2 -8094.748} C_VEL
LIN {X 0,Y 460.823,Z 136.081,A -85,B 0,C 180,E1 -8097.377,E2 -8097.377} C_VEL
LIN {X 0,Y 460.852,Z 136.075,A -85,B 0,C 180,E1 -8100,E2 -8100} C_VEL
LIN {X 0,Y 460.823,Z 136.084,A -85,B 0,C 180,E1 -8102.622,E2 -8102.622} C_VEL
LIN {X 0,Y 460.7,Z 136.095,A -85,B 0,C 180,E1 -8106.13,E2 -8106.13} C_VEL
LIN {X 0,Y 460.626,Z 136.109,A -85,B 0,C 180,E1 -8108.776,E2 -8108.776} C_VEL
LIN {X 0,Y 460.61,Z 136.111,A -85,B 0,C 180,E1 -8112.444,E2 -8112.444} C_VEL
LIN {X 0,Y 460.597,Z 136.108,A -85,B 0,C 180,E1 -8115.997,E2 -8115.997} C_VEL
LIN {X 0,Y 460.568,Z 136.113,A -85,B 0,C 180,E1 -8118.902,E2 -8118.902} C_VEL
LIN {X 0,Y 460.512,Z 136.117,A -85,B 0,C 180,E1 -8121.485,E2 -8121.485} C_VEL
LIN {X 0,Y 460.538,Z 136.122,A -85,B 0,C 180,E1 -8124.332,E2 -8124.332} C_VEL
LIN {X 0,Y 460.58,Z 136.109,A -85,B 0,C 180,E1 -8127.243,E2 -8127.243} C_VEL
LIN {X 0,Y 460.507,Z 136.126,A -85,B 0,C 180,E1 -8130.24,E2 -8130.24} C_VEL
LIN {X 0,Y 460.525,Z 136.116,A -85,B 0,C 180,E1 -8133.325,E2 -8133.325} C_VEL
LIN {X 0,Y 460.475,Z 136.124,A -85,B 0,C 180,E1 -8136.529,E2 -8136.529} C_VEL
LIN {X 0,Y 460.574,Z 136.115,A -85,B 0,C 180,E1 -8139.857,E2 -8139.857} C_VEL
LIN {X 0,Y 460.537,Z 136.114,A -85,B 0,C 180,E1 -8142.904,E2 -8142.904} C_VEL
LIN {X 0,Y 460.519,Z 136.123,A -85,B 0,C 180,E1 -8145.829,E2 -8145.829} C_VEL
LIN {X 0,Y 460.538,Z 136.114,A -85,B 0,C 180,E1 -8148.99,E2 -8148.99} C_VEL
LIN {X 0,Y 460.542,Z 136.115,A -85,B 0,C 180,E1 -8151.269,E2 -8151.269} C_VEL
LIN {X 0,Y 460.508,Z 136.118,A -85,B 0,C 180,E1 -8154.555,E2 -8154.555} C_VEL
LIN {X 0,Y 460.527,Z 136.123,A -85,B 0,C 180,E1 -8157.716,E2 -8157.716} C_VEL
LIN {X 0,Y 460.535,Z 136.114,A -85,B 0,C 180,E1 -8160.769,E2 -8160.769} C_VEL
LIN {X 0,Y 460.564,Z 136.116,A -85,B 0,C 180,E1 -8163.735,E2 -8163.735} C_VEL
LIN {X 0,Y 460.541,Z 136.114,A -85,B 0,C 180,E1 -8166.624,E2 -8166.624} C_VEL
LIN {X 0,Y 460.548,Z 136.12,A -85,B 0,C 180,E1 -8169.453,E2 -8169.453} C_VEL
LIN {X 0,Y 460.555,Z 136.112,A -85,B 0,C 180,E1 -8172.23,E2 -8172.23} C_VEL
LIN {X 0,Y 460.563,Z 136.114,A -85,B 0,C 180,E1 -8174.965,E2 -8174.965} C_VEL
LIN {X 0,Y 460.608,Z 136.106,A -85,B 0,C 180,E1 -8178.56,E2 -8178.56} C_VEL
LIN {X 0,Y 460.574,Z 136.112,A -85,B 0,C 180,E1 -8179.225,E2 -8179.225} C_VEL
LIN {X 0,Y 459.92,Z 136.199,A -85,B 0,C 180,E1 -8179.955,E2 -8179.955} C_VEL
LIN {X 0,Y 457.102,Z 136.553,A -85,B 0,C 180,E1 -8181.141,E2 -8181.141} C_VEL
LIN {X 0,Y 454.722,Z 136.847,A -85,B 0,C 180,E1 -8182.098,E2 -8182.098} C_VEL
LIN {X 0,Y 453.711,Z 136.969,A -85,B 0,C 180,E1 -8182.837,E2 -8182.837} C_VEL
LIN {X 0,Y 453.634,Z 136.976,A -85,B 0,C 180,E1 -8183.087,E2 -8183.087} C_VEL
LIN {X 0,Y 453.669,Z 136.972,A -85,B 0,C 180,E1 -8184.667,E2 -8184.667} C_VEL
LIN {X 0,Y 453.762,Z 136.962,A -85,B 0,C 180,E1 -8187.337,E2 -8187.337} C_VEL
LIN {X 0,Y 453.821,Z 136.951,A -85,B 0,C 180,E1 -8190.001,E2 -8190.001} C_VEL
LIN {X 0,Y 453.762,Z 136.962,A -85,B 0,C 180,E1 -8192.664,E2 -8192.664} C_VEL
LIN {X 0,Y 453.676,Z 136.97,A -85,B 0,C 180,E1 -8196.226,E2 -8196.226} C_VEL
LIN {X 0,Y 453.59,Z 136.986,A -85,B 0,C 180,E1 -8198.914,E2 -8198.914} C_VEL
LIN {X 0,Y 453.561,Z 136.988,A -85,B 0,C 180,E1 -8202.529,E2 -8202.529} C_VEL
LIN {X 0,Y 453.538,Z 136.992,A -85,B 0,C 180,E1 -8206.197,E2 -8206.197} C_VEL
LIN {X 0,Y 453.547,Z 136.994,A -85,B 0,C 180,E1 -8207.53,E2 -8207.53} C_VEL
LIN {X 0,Y 454.621,Z 143.259,A -85,B 0,C 180,E1 -8208.944,E2 -8208.944} C_VEL
LIN {X 0,Y 454.614,Z 150.799,A -85,B 0,C 180,E1 -8210.562,E2 -8210.562} C_VEL
LIN {X 0,Y 457.698,Z 166.2,A -85,B 0,C 180,E1 -8210.946,E2 -8210.946} C_VEL
LIN {X 0,Y 456.711,Z 258.51,A -85,B 0,C 180,E1 -8212.463,E2 -8212.463} C_VEL
LIN {X 0,Y 456.44,Z 272.131,A -85,B 0,C 180,E1 -8212.879,E2 -8212.879} C_VEL
LIN {X 0,Y 456.101,Z 284.474,A -85,B 0,C 180,E1 -8213.438,E2 -8213.438} C_VEL
LIN {X 0,Y 455.751,Z 295.545,A -85,B 0,C 180,E1 -8214.11,E2 -8214.11} C_VEL
LIN {X 0,Y 455.154,Z 307.123,A -85,B 0,C 180,E1 -8215.005,E2 -8215.005} C_VEL
LIN {X 0,Y 454.607,Z 317.711,A -85,B 0,C 180,E1 -8216.034,E2 -8216.034} C_VEL
LIN {X 0,Y 454.134,Z 327.055,A -85,B 0,C 180,E1 -8217.164,E2 -8217.164} C_VEL
LIN {X 0,Y 453.65,Z 336.077,A -85,B 0,C 180,E1 -8218.516,E2 -8218.516} C_VEL
LIN {X 0,Y 453.31,Z 342.737,A -85,B 0,C 180,E1 -8219.75,E2 -8219.75} C_VEL
LIN {X 0,Y 452.998,Z 348.652,A -85,B 0,C 180,E1 -8221.105,E2 -8221.105} C_VEL
LIN {X 0,Y 452.796,Z 353.033,A -85,B 0,C 180,E1 -8222.377,E2 -8222.377} C_VEL
LIN {X 0,Y 452.6,Z 357.172,A -85,B 0,C 180,E1 -8223.988,E2 -8223.988} C_VEL
LIN {X 0,Y 452.466,Z 359.166,A -85,B 0,C 180,E1 -8225.08,E2 -8225.08} C_VEL
LIN {X 0,Y 452.432,Z 360.525,A -85,B 0,C 180,E1 -8226.178,E2 -8226.178} C_VEL
LIN {X 0,Y 452.404,Z 361.392,A -85,B 0,C 180,E1 -8227.603,E2 -8227.603} C_VEL
LIN {X 0,Y 452.395,Z 361.238,A -85,B 0,C 180,E1 -8229.037,E2 -8229.037} C_VEL
LIN {X 0,Y 452.492,Z 359.741,A -85,B 0,C 180,E1 -8230.719,E2 -8230.719} C_VEL
LIN {X 0,Y 452.693,Z 356.596,A -85,B 0,C 180,E1 -8232.481,E2 -8232.481} C_VEL
LIN {X 0,Y 452.826,Z 353.477,A -85,B 0,C 180,E1 -8233.686,E2 -8233.686} C_VEL
LIN {X 0,Y 453.071,Z 348.113,A -85,B 0,C 180,E1 -8235.235,E2 -8235.235} C_VEL
LIN {X 0,Y 453.441,Z 341.24,A -85,B 0,C 180,E1 -8236.759,E2 -8236.759} C_VEL
LIN {X 0,Y 453.847,Z 334.124,A -85,B 0,C 180,E1 -8238.014,E2 -8238.014} C_VEL
LIN {X 0,Y 454.351,Z 325.188,A -85,B 0,C 180,E1 -8239.284,E2 -8239.284} C_VEL
LIN {X 0,Y 454.887,Z 315.867,A -85,B 0,C 180,E1 -8240.361,E2 -8240.361} C_VEL
LIN {X 0,Y 455.356,Z 305.776,A -85,B 0,C 180,E1 -8241.313,E2 -8241.313} C_VEL
LIN {X 0,Y 455.998,Z 294.607,A -85,B 0,C 180,E1 -8242.15,E2 -8242.15} C_VEL
LIN {X 0,Y 456.437,Z 283.162,A -85,B 0,C 180,E1 -8242.818,E2 -8242.818} C_VEL
LIN {X 0,Y 456.735,Z 269.949,A -85,B 0,C 180,E1 -8243.39,E2 -8243.39} C_VEL
LIN {X 0,Y 457.008,Z 257.268,A -85,B 0,C 180,E1 -8243.748,E2 -8243.748} C_VEL
LIN {X 0,Y 457.937,Z 166.102,A -85,B 0,C 180,E1 -8245.254,E2 -8245.254} C_VEL
LIN {X 0,Y 454.793,Z 151.292,A -85,B 0,C 180,E1 -8245.665,E2 -8245.665} C_VEL
LIN {X 0,Y 454.786,Z 143.666,A -85,B 0,C 180,E1 -8247.258,E2 -8247.258} C_VEL
LIN {X 0,Y 453.505,Z 136.997,A -85,B 0,C 180,E1 -8248.751,E2 -8248.751} C_VEL
LIN {X 0,Y 453.535,Z 136.991,A -85,B 0,C 180,E1 -8252.298,E2 -8252.298} C_VEL
LIN {X 0,Y 453.498,Z 137.002,A -85,B 0,C 180,E1 -8255.265,E2 -8255.265} C_VEL
LIN {X 0,Y 453.484,Z 136.998,A -85,B 0,C 180,E1 -8258.416,E2 -8258.416} C_VEL
LIN {X 0,Y 453.526,Z 136.994,A -85,B 0,C 180,E1 -8261.009,E2 -8261.009} C_VEL
LIN {X 0,Y 453.573,Z 136.984,A -85,B 0,C 180,E1 -8263.88,E2 -8263.88} C_VEL
LIN {X 0,Y 453.568,Z 136.987,A -85,B 0,C 180,E1 -8267.472,E2 -8267.472} C_VEL
LIN {X 0,Y 453.588,Z 136.985,A -85,B 0,C 180,E1 -8271.087,E2 -8271.087} C_VEL
LIN {X 0,Y 453.642,Z 136.976,A -85,B 0,C 180,E1 -8273.775,E2 -8273.775} C_VEL
LIN {X 0,Y 453.709,Z 136.967,A -85,B 0,C 180,E1 -8277.337,E2 -8277.337} C_VEL
LIN {X 0,Y 453.772,Z 136.958,A -85,B 0,C 180,E1 -8280,E2 -8280} C_VEL
LIN {X 0,Y 453.706,Z 136.964,A -85,B 0,C 180,E1 -8282.664,E2 -8282.664} C_VEL
LIN {X 0,Y 453.639,Z 136.973,A -85,B 0,C 180,E1 -8286.226,E2 -8286.226} C_VEL
LIN {X 0,Y 453.56,Z 136.984,A -85,B 0,C 180,E1 -8288.914,E2 -8288.914} C_VEL
LIN {X 0,Y 453.57,Z 136.983,A -85,B 0,C 180,E1 -8292.529,E2 -8292.529} C_VEL
LIN {X 0,Y 453.49,Z 136.994,A -85,B 0,C 180,E1 -8296.198,E2 -8296.198} C_VEL
LIN {X 0,Y 453.464,Z 136.996,A -85,B 0,C 180,E1 -8299.018,E2 -8299.018} C_VEL
LIN {X 0,Y 453.471,Z 136.998,A -85,B 0,C 180,E1 -8301.837,E2 -8301.837} C_VEL
LIN {X 0,Y 453.454,Z 136.996,A -85,B 0,C 180,E1 -8304.738,E2 -8304.738} C_VEL
LIN {X 0,Y 453.46,Z 136.994,A -85,B 0,C 180,E1 -8307.941,E2 -8307.941} C_VEL
LIN {X 0,Y 453.451,Z 137.001,A -85,B 0,C 180,E1 -8310.762,E2 -8310.762} C_VEL
LIN {X 0,Y 453.471,Z 136.995,A -85,B 0,C 180,E1 -8313.914,E2 -8313.914} C_VEL
LIN {X 0,Y 453.454,Z 137,A -85,B 0,C 180,E1 -8317.19,E2 -8317.19} C_VEL
LIN {X 0,Y 453.475,Z 137.001,A -85,B 0,C 180,E1 -8320.612,E2 -8320.612} C_VEL
LIN {X 0,Y 453.486,Z 136.999,A -85,B 0,C 180,E1 -8324.528,E2 -8324.528} C_VEL
LIN {X 0,Y 453.454,Z 137.003,A -85,B 0,C 180,E1 -8328.069,E2 -8328.069} C_VEL
LIN {X 0,Y 453.453,Z 137.002,A -85,B 0,C 180,E1 -8330.8,E2 -8330.8} C_VEL
LIN {X 0,Y 453.456,Z 137.002,A -85,B 0,C 180,E1 -8333.917,E2 -8333.917} C_VEL
LIN {X 0,Y 453.488,Z 136.999,A -85,B 0,C 180,E1 -8337.151,E2 -8337.151} C_VEL
LIN {X 0,Y 453.472,Z 137.003,A -85,B 0,C 180,E1 -8340.267,E2 -8340.267} C_VEL
LIN {X 0,Y 453.541,Z 137.037,A -85,B 0,C 180,E1 -8343.171,E2 -8343.171} C_VEL
LIN {X 0,Y 455.88,Z 148.955,A -85,B 0,C 180,E1 -8345.446,E2 -8345.446} C_VEL
LIN {X 0,Y 455.674,Z 156.878,A -85,B 0,C 180,E1 -8346.84,E2 -8346.84} C_VEL
LIN {X 0,Y 454.881,Z 174.521,A -85,B 0,C 180,E1 -8349.893,E2 -8349.893} C_VEL
LIN {X 0,Y 454.307,Z 189.045,A -85,B 0,C 180,E1 -8352.371,E2 -8352.371} C_VEL
LIN {X 0,Y 457.619,Z 211.314,A -85,B 0,C 180,E1 -8352.882,E2 -8352.882} C_VEL
LIN {X 0,Y 456.801,Z 298.243,A -85,B 0,C 180,E1 -8354.323,E2 -8354.323} C_VEL
LIN {X 0,Y 456.377,Z 311.311,A -85,B 0,C 180,E1 -8354.709,E2 -8354.709} C_VEL
LIN {X 0,Y 455.821,Z 323.977,A -85,B 0,C 180,E1 -8355.261,E2 -8355.261} C_VEL
LIN {X 0,Y 455.283,Z 335.279,A -85,B 0,C 180,E1 -8355.928,E2 -8355.928} C_VEL
LIN {X 0,Y 454.705,Z 347.215,A -85,B 0,C 180,E1 -8356.841,E2 -8356.841} C_VEL
LIN {X 0,Y 454.129,Z 357.531,A -85,B 0,C 180,E1 -8357.827,E2 -8357.827} C_VEL
LIN {X 0,Y 453.73,Z 366.167,A -85,B 0,C 180,E1 -8358.836,E2 -8358.836} C_VEL
LIN {X 0,Y 453.265,Z 374.137,A -85,B 0,C 180,E1 -8359.954,E2 -8359.954} C_VEL
LIN {X 0,Y 452.916,Z 381.931,A -85,B 0,C 180,E1 -8361.298,E2 -8361.298} C_VEL
LIN {X 0,Y 452.67,Z 389.123,A -85,B 0,C 180,E1 -8362.865,E2 -8362.865} C_VEL
LIN {X 0,Y 452.526,Z 393.912,A -85,B 0,C 180,E1 -8364.206,E2 -8364.206} C_VEL
LIN {X 0,Y 452.487,Z 397.576,A -85,B 0,C 180,E1 -8365.545,E2 -8365.545} C_VEL
LIN {X 0,Y 452.494,Z 399.468,A -85,B 0,C 180,E1 -8366.438,E2 -8366.438} C_VEL
LIN {X 0,Y 452.528,Z 400.888,A -85,B 0,C 180,E1 -8367.329,E2 -8367.329} C_VEL
LIN {X 0,Y 452.494,Z 402.526,A -85,B 0,C 180,E1 -8369.11,E2 -8369.11} C_VEL
LIN {X 0,Y 452.475,Z 402.743,A -85,B 0,C 180,E1 -8369.999,E2 -8369.999} C_VEL
LIN {X 0,Y 452.494,Z 402.524,A -85,B 0,C 180,E1 -8370.889,E2 -8370.889} C_VEL
LIN {X 0,Y 452.528,Z 400.905,A -85,B 0,C 180,E1 -8372.67,E2 -8372.67} C_VEL
LIN {X 0,Y 452.494,Z 399.478,A -85,B 0,C 180,E1 -8373.561,E2 -8373.561} C_VEL
LIN {X 0,Y 452.541,Z 396.498,A -85,B 0,C 180,E1 -8374.899,E2 -8374.899} C_VEL
LIN {X 0,Y 452.569,Z 392.074,A -85,B 0,C 180,E1 -8376.347,E2 -8376.347} C_VEL
LIN {X 0,Y 452.758,Z 386.229,A -85,B 0,C 180,E1 -8377.806,E2 -8377.806} C_VEL
LIN {X 0,Y 453.033,Z 379.439,A -85,B 0,C 180,E1 -8379.149,E2 -8379.149} C_VEL
LIN {X 0,Y 453.403,Z 371.004,A -85,B 0,C 180,E1 -8380.493,E2 -8380.493} C_VEL
LIN {X 0,Y 453.89,Z 362.314,A -85,B 0,C 180,E1 -8381.612,E2 -8381.612} C_VEL
LIN {X 0,Y 454.386,Z 352.02,A -85,B 0,C 180,E1 -8382.693,E2 -8382.693} C_VEL
LIN {X 0,Y 454.94,Z 340.982,A -85,B 0,C 180,E1 -8383.626,E2 -8383.626} C_VEL
LIN {X 0,Y 455.515,Z 329.164,A -85,B 0,C 180,E1 -8384.405,E2 -8384.405} C_VEL
LIN {X 0,Y 456.05,Z 316.898,A -85,B 0,C 180,E1 -8385.016,E2 -8385.016} C_VEL
LIN {X 0,Y 456.46,Z 304.413,A -85,B 0,C 180,E1 -8385.459,E2 -8385.459} C_VEL
LIN {X 0,Y 456.693,Z 291.835,A -85,B 0,C 180,E1 -8385.737,E2 -8385.737} C_VEL
LIN {X 0,Y 457.413,Z 211.356,A -85,B 0,C 180,E1 -8387.039,E2 -8387.039} C_VEL
LIN {X 0,Y 454.295,Z 189.832,A -85,B 0,C 180,E1 -8387.52,E2 -8387.52} C_VEL
LIN {X 0,Y 454.992,Z 173.512,A -85,B 0,C 180,E1 -8390.337,E2 -8390.337} C_VEL
LIN {X 0,Y 456.034,Z 153.341,A -85,B 0,C 180,E1 -8393.862,E2 -8393.862} C_VEL
LIN {X 0,Y 455.976,Z 149.278,A -85,B 0,C 180,E1 -8394.591,E2 -8394.591} C_VEL
LIN {X 0,Y 453.557,Z 136.99,A -85,B 0,C 180,E1 -8396.951,E2 -8396.951} C_VEL
LIN {X 0,Y 453.473,Z 137,A -85,B 0,C 180,E1 -8399.784,E2 -8399.784} C_VEL
LIN {X 0,Y 453.491,Z 136.992,A -85,B 0,C 180,E1 -8403.189,E2 -8403.189} C_VEL
LIN {X 0,Y 453.454,Z 137,A -85,B 0,C 180,E1 -8406.298,E2 -8406.298} C_VEL
LIN {X 0,Y 453.517,Z 136.991,A -85,B 0,C 180,E1 -8409.446,E2 -8409.446} C_VEL
LIN {X 0,Y 453.461,Z 136.996,A -85,B 0,C 180,E1 -8412.995,E2 -8412.995} C_VEL
LIN {X 0,Y 453.464,Z 137.003,A -85,B 0,C 180,E1 -8415.778,E2 -8415.778} C_VEL
LIN {X 0,Y 453.479,Z 136.995,A -85,B 0,C 180,E1 -8418.209,E2 -8418.209} C_VEL
LIN {X 0,Y 453.487,Z 136.992,A -85,B 0,C 180,E1 -8420.794,E2 -8420.794} C_VEL
LIN {X 0,Y 453.453,Z 137,A -85,B 0,C 180,E1 -8423.917,E2 -8423.917} C_VEL
LIN {X 0,Y 453.478,Z 136.997,A -85,B 0,C 180,E1 -8427.15,E2 -8427.15} C_VEL
LIN {X 0,Y 453.473,Z 136.994,A -85,B 0,C 180,E1 -8430.268,E2 -8430.268} C_VEL
LIN {X 0,Y 453.506,Z 136.997,A -85,B 0,C 180,E1 -8433.293,E2 -8433.293} C_VEL
LIN {X 0,Y 453.502,Z 136.99,A -85,B 0,C 180,E1 -8436.238,E2 -8436.238} C_VEL
LIN {X 0,Y 453.482,Z 136.999,A -85,B 0,C 180,E1 -8439.117,E2 -8439.117} C_VEL
LIN {X 0,Y 453.502,Z 136.991,A -85,B 0,C 180,E1 -8441.944,E2 -8441.944} C_VEL
LIN {X 0,Y 453.539,Z 136.988,A -85,B 0,C 180,E1 -8444.726,E2 -8444.726} C_VEL
LIN {X 0,Y 453.558,Z 136.984,A -85,B 0,C 180,E1 -8448.378,E2 -8448.378} C_VEL
LIN {X 0,Y 453.65,Z 136.972,A -85,B 0,C 180,E1 -8451.985,E2 -8451.985} C_VEL
LIN {X 0,Y 453.666,Z 136.974,A -85,B 0,C 180,E1 -8454.666,E2 -8454.666} C_VEL
LIN {X 0,Y 453.763,Z 136.96,A -85,B 0,C 180,E1 -8457.336,E2 -8457.336} C_VEL
LIN {X 0,Y 453.822,Z 136.951,A -85,B 0,C 180,E1 -8460,E2 -8460} C_VEL
LIN {X 0,Y 453.763,Z 136.964,A -85,B 0,C 180,E1 -8462.663,E2 -8462.663} C_VEL
LIN {X 0,Y 453.668,Z 136.972,A -85,B 0,C 180,E1 -8466.225,E2 -8466.225} C_VEL
LIN {X 0,Y 453.59,Z 136.984,A -85,B 0,C 180,E1 -8468.913,E2 -8468.913} C_VEL
LIN {X 0,Y 453.56,Z 136.99,A -85,B 0,C 180,E1 -8472.528,E2 -8472.528} C_VEL
LIN {X 0,Y 453.541,Z 136.989,A -85,B 0,C 180,E1 -8476.195,E2 -8476.195} C_VEL
LIN {X 0,Y 453.517,Z 136.99,A -85,B 0,C 180,E1 -8479.041,E2 -8479.041} C_VEL
LIN {X 0,Y 453.473,Z 136.996,A -85,B 0,C 180,E1 -8481.836,E2 -8481.836} C_VEL
LIN {X 0,Y 453.51,Z 136.992,A -85,B 0,C 180,E1 -8484.734,E2 -8484.734} C_VEL
LIN {X 0,Y 453.533,Z 136.99,A -85,B 0,C 180,E1 -8487.961,E2 -8487.961} C_VEL
LIN {X 0,Y 453.462,Z 136.996,A -85,B 0,C 180,E1 -8491.525,E2 -8491.525} C_VEL
LIN {X 0,Y 453.484,Z 136.994,A -85,B 0,C 180,E1 -8494.777,E2 -8494.777} C_VEL
LIN {X 0,Y 453.481,Z 136.998,A -85,B 0,C 180,E1 -8498.309,E2 -8498.309} C_VEL
LIN {X 0,Y 453.511,Z 136.991,A -85,B 0,C 180,E1 -8500.606,E2 -8500.606} C_VEL
LIN {X 0,Y 453.477,Z 136.994,A -85,B 0,C 180,E1 -8503.248,E2 -8503.248} C_VEL
LIN {X 0,Y 453.472,Z 137,A -85,B 0,C 180,E1 -8505.78,E2 -8505.78} C_VEL
LIN {X 0,Y 453.491,Z 136.995,A -85,B 0,C 180,E1 -8508.211,E2 -8508.211} C_VEL
LIN {X 0,Y 453.528,Z 136.987,A -85,B 0,C 180,E1 -8510.787,E2 -8510.787} C_VEL
LIN {X 0,Y 453.452,Z 137.002,A -85,B 0,C 180,E1 -8513.918,E2 -8513.918} C_VEL
LIN {X 0,Y 453.478,Z 136.995,A -85,B 0,C 180,E1 -8517.151,E2 -8517.151} C_VEL
LIN {X 0,Y 453.47,Z 136.995,A -85,B 0,C 180,E1 -8520.269,E2 -8520.269} C_VEL
LIN {X 0,Y 453.509,Z 136.994,A -85,B 0,C 180,E1 -8523.295,E2 -8523.295} C_VEL
LIN {X 0,Y 453.499,Z 136.991,A -85,B 0,C 180,E1 -8526.239,E2 -8526.239} C_VEL
LIN {X 0,Y 453.479,Z 136.997,A -85,B 0,C 180,E1 -8529.118,E2 -8529.118} C_VEL
LIN {X 0,Y 453.507,Z 136.991,A -85,B 0,C 180,E1 -8531.945,E2 -8531.945} C_VEL
LIN {X 0,Y 453.537,Z 136.987,A -85,B 0,C 180,E1 -8534.727,E2 -8534.727} C_VEL
LIN {X 0,Y 453.556,Z 136.984,A -85,B 0,C 180,E1 -8538.379,E2 -8538.379} C_VEL
LIN {X 0,Y 453.648,Z 136.972,A -85,B 0,C 180,E1 -8541.986,E2 -8541.986} C_VEL
LIN {X 0,Y 453.634,Z 136.976,A -85,B 0,C 180,E1 -8543.087,E2 -8543.087} C_VEL
LIN {X 0,Y 452.949,Z 137.062,A -85,B 0,C 180,E1 -8543.828,E2 -8543.828} C_VEL
LIN {X 0,Y 450,Z 137.434,A -85,B 0,C 180,E1 -8545.03,E2 -8545.03} C_VEL
LIN {X 0,Y 447.576,Z 137.731,A -85,B 0,C 180,E1 -8545.999,E2 -8545.999} C_VEL
LIN {X 0,Y 446.639,Z 137.849,A -85,B 0,C 180,E1 -8546.75,E2 -8546.75} C_VEL
LIN {X 0,Y 446.619,Z 137.85,A -85,B 0,C 180,E1 -8547.003,E2 -8547.003} C_VEL
LIN {X 0,Y 446.791,Z 137.826,A -85,B 0,C 180,E1 -8550.001,E2 -8550.001} C_VEL
LIN {X 0,Y 446.706,Z 137.842,A -85,B 0,C 180,E1 -8552.706,E2 -8552.706} C_VEL
LIN {X 0,Y 446.645,Z 137.846,A -85,B 0,C 180,E1 -8556.324,E2 -8556.324} C_VEL
LIN {X 0,Y 446.536,Z 137.863,A -85,B 0,C 180,E1 -8559.056,E2 -8559.056} C_VEL
LIN {X 0,Y 446.519,Z 137.868,A -85,B 0,C 180,E1 -8562.73,E2 -8562.73} C_VEL
LIN {X 0,Y 446.516,Z 137.867,A -85,B 0,C 180,E1 -8566.238,E2 -8566.238} C_VEL
LIN {X 0,Y 446.512,Z 137.959,A -85,B 0,C 180,E1 -8567.372,E2 -8567.372} C_VEL
LIN {X 0,Y 447.693,Z 145.156,A -85,B 0,C 180,E1 -8569.011,E2 -8569.011} C_VEL
LIN {X 0,Y 447.684,Z 151.271,A -85,B 0,C 180,E1 -8570.307,E2 -8570.307} C_VEL
LIN {X 0,Y 450.927,Z 167.549,A -85,B 0,C 180,E1 -8570.712,E2 -8570.712} C_VEL
LIN {X 0,Y 449.886,Z 258.198,A -85,B 0,C 180,E1 -8572.22,E2 -8572.22} C_VEL
LIN {X 0,Y 449.561,Z 271.939,A -85,B 0,C 180,E1 -8572.639,E2 -8572.639} C_VEL
LIN {X 0,Y 449.237,Z 284.434,A -85,B 0,C 180,E1 -8573.207,E2 -8573.207} C_VEL
LIN {X 0,Y 448.834,Z 295.778,A -85,B 0,C 180,E1 -8573.902,E2 -8573.902} C_VEL
LIN {X 0,Y 448.236,Z 307.067,A -85,B 0,C 180,E1 -8574.784,E2 -8574.784} C_VEL
LIN {X 0,Y 447.671,Z 317.712,A -85,B 0,C 180,E1 -8575.827,E2 -8575.827} C_VEL
LIN {X 0,Y 447.189,Z 326.799,A -85,B 0,C 180,E1 -8576.929,E2 -8576.929} C_VEL
LIN {X 0,Y 446.685,Z 335.482,A -85,B 0,C 180,E1 -8578.228,E2 -8578.228} C_VEL
LIN {X 0,Y 446.299,Z 342.834,A -85,B 0,C 180,E1 -8579.588,E2 -8579.588} C_VEL
LIN {X 0,Y 445.934,Z 349.222,A -85,B 0,C 180,E1 -8581.075,E2 -8581.075} C_VEL
LIN {X 0,Y 445.701,Z 353.719,A -85,B 0,C 180,E1 -8582.421,E2 -8582.421} C_VEL
LIN {X 0,Y 445.508,Z 357.735,A -85,B 0,C 180,E1 -8584.058,E2 -8584.058} C_VEL
LIN {X 0,Y 445.359,Z 360.393,A -85,B 0,C 180,E1 -8585.725,E2 -8585.725} C_VEL
LIN {X 0,Y 445.311,Z 361.393,A -85,B 0,C 180,E1 -8586.851,E2 -8586.851} C_VEL
LIN {X 0,Y 445.322,Z 361.791,A -85,B 0,C 180,E1 -8587.988,E2 -8587.988} C_VEL
LIN {X 0,Y 445.306,Z 361.42,A -85,B 0,C 180,E1 -8589.346,E2 -8589.346} C_VEL
LIN {X 0,Y 445.416,Z 360.071,A -85,B 0,C 180,E1 -8590.768,E2 -8590.768} C_VEL
LIN {X 0,Y 445.578,Z 357.775,A -85,B 0,C 180,E1 -8592.157,E2 -8592.157} C_VEL
LIN {X 0,Y 445.723,Z 354.57,A -85,B 0,C 180,E1 -8593.506,E2 -8593.506} C_VEL
LIN {X 0,Y 445.927,Z 350.408,A -85,B 0,C 180,E1 -8594.829,E2 -8594.829} C_VEL
LIN {X 0,Y 446.307,Z 343.946,A -85,B 0,C 180,E1 -8596.417,E2 -8596.417} C_VEL
LIN {X 0,Y 446.788,Z 335.897,A -85,B 0,C 180,E1 -8597.936,E2 -8597.936} C_VEL
LIN {X 0,Y 447.241,Z 328.012,A -85,B 0,C 180,E1 -8599.137,E2 -8599.137} C_VEL
LIN {X 0,Y 447.845,Z 318.21,A -85,B 0,C 180,E1 -8600.349,E2 -8600.349} C_VEL
LIN {X 0,Y 448.379,Z 307.479,A -85,B 0,C 180,E1 -8601.409,E2 -8601.409} C_VEL
LIN {X 0,Y 449.073,Z 296.2,A -85,B 0,C 180,E1 -8602.293,E2 -8602.293} C_VEL
LIN {X 0,Y 449.541,Z 285.064,A -85,B 0,C 180,E1 -8602.978,E2 -8602.978} C_VEL
LIN {X 0,Y 449.85,Z 271.78,A -85,B 0,C 180,E1 -8603.583,E2 -8603.583} C_VEL
LIN {X 0,Y 450.196,Z 258.505,A -85,B 0,C 180,E1 -8603.982,E2 -8603.982} C_VEL
LIN {X 0,Y 451.214,Z 167.038,A -85,B 0,C 180,E1 -8605.523,E2 -8605.523} C_VEL
LIN {X 0,Y 447.903,Z 151.64,A -85,B 0,C 180,E1 -8605.962,E2 -8605.962} C_VEL
LIN {X 0,Y 447.915,Z 145.641,A -85,B 0,C 180,E1 -8607.227,E2 -8607.227} C_VEL
LIN {X 0,Y 446.441,Z 137.877,A -85,B 0,C 180,E1 -8608.966,E2 -8608.966} C_VEL
LIN {X 0,Y 446.487,Z 137.871,A -85,B 0,C 180,E1 -8611.822,E2 -8611.822} C_VEL
LIN {X 0,Y 446.442,Z 137.879,A -85,B 0,C 180,E1 -8614.847,E2 -8614.847} C_VEL
LIN {X 0,Y 446.451,Z 137.874,A -85,B 0,C 180,E1 -8618.246,E2 -8618.246} C_VEL
LIN {X 0,Y 446.454,Z 137.871,A -85,B 0,C 180,E1 -8621.65,E2 -8621.65} C_VEL
LIN {X 0,Y 446.511,Z 137.867,A -85,B 0,C 180,E1 -8624.48,E2 -8624.48} C_VEL
LIN {X 0,Y 446.521,Z 137.866,A -85,B 0,C 180,E1 -8628.194,E2 -8628.194} C_VEL
LIN {X 0,Y 446.535,Z 137.865,A -85,B 0,C 180,E1 -8630.945,E2 -8630.945} C_VEL
LIN {X 0,Y 446.612,Z 137.852,A -85,B 0,C 180,E1 -8633.676,E2 -8633.676} C_VEL
LIN {X 0,Y 446.658,Z 137.845,A -85,B 0,C 180,E1 -8637.295,E2 -8637.295} C_VEL
LIN {X 0,Y 446.722,Z 137.836,A -85,B 0,C 180,E1 -8640,E2 -8640} C_VEL
LIN {X 0,Y 446.656,Z 137.841,A -85,B 0,C 180,E1 -8642.706,E2 -8642.706} C_VEL
LIN {X 0,Y 446.609,Z 137.848,A -85,B 0,C 180,E1 -8646.325,E2 -8646.325} C_VEL
LIN {X 0,Y 446.511,Z 137.862,A -85,B 0,C 180,E1 -8649.056,E2 -8649.056} C_VEL
LIN {X 0,Y 446.497,Z 137.863,A -85,B 0,C 180,E1 -8652.731,E2 -8652.731} C_VEL
LIN {X 0,Y 446.459,Z 137.869,A -85,B 0,C 180,E1 -8656.209,E2 -8656.209} C_VEL
LIN {X 0,Y 446.405,Z 137.876,A -85,B 0,C 180,E1 -8659.307,E2 -8659.307} C_VEL
LIN {X 0,Y 446.408,Z 137.875,A -85,B 0,C 180,E1 -8662.201,E2 -8662.201} C_VEL
LIN {X 0,Y 446.411,Z 137.878,A -85,B 0,C 180,E1 -8665.156,E2 -8665.156} C_VEL
LIN {X 0,Y 446.42,Z 137.871,A -85,B 0,C 180,E1 -8668.184,E2 -8668.184} C_VEL
LIN {X 0,Y 446.396,Z 137.877,A -85,B 0,C 180,E1 -8671.302,E2 -8671.302} C_VEL
LIN {X 0,Y 446.427,Z 137.875,A -85,B 0,C 180,E1 -8674.524,E2 -8674.524} C_VEL
LIN {X 0,Y 446.415,Z 137.873,A -85,B 0,C 180,E1 -8678.078,E2 -8678.078} C_VEL
LIN {X 0,Y 446.405,Z 137.876,A -85,B 0,C 180,E1 -8681.394,E2 -8681.394} C_VEL
LIN {X 0,Y 446.454,Z 137.874,A -85,B 0,C 180,E1 -8685.104,E2 -8685.104} C_VEL
LIN {X 0,Y 446.412,Z 137.881,A -85,B 0,C 180,E1 -8688.606,E2 -8688.606} C_VEL
LIN {X 0,Y 446.415,Z 137.879,A -85,B 0,C 180,E1 -8691.921,E2 -8691.921} C_VEL
LIN {X 0,Y 446.433,Z 137.874,A -85,B 0,C 180,E1 -8695.477,E2 -8695.477} C_VEL
LIN {X 0,Y 446.42,Z 137.879,A -85,B 0,C 180,E1 -8698.699,E2 -8698.699} C_VEL
LIN {X 0,Y 446.455,Z 137.876,A -85,B 0,C 180,E1 -8701.83,E2 -8701.83} C_VEL
LIN {X 0,Y 446.492,Z 137.969,A -85,B 0,C 180,E1 -8702.93,E2 -8702.93} C_VEL
LIN {X 0,Y 448.89,Z 149.825,A -85,B 0,C 180,E1 -8705.241,E2 -8705.241} C_VEL
LIN {X 0,Y 448.962,Z 155.262,A -85,B 0,C 180,E1 -8706.228,E2 -8706.228} C_VEL
LIN {X 0,Y 447.916,Z 175.627,A -85,B 0,C 180,E1 -8709.806,E2 -8709.806} C_VEL
LIN {X 0,Y 447.344,Z 188.639,A -85,B 0,C 180,E1 -8712.068,E2 -8712.068} C_VEL
LIN {X 0,Y 450.857,Z 212.973,A -85,B 0,C 180,E1 -8712.639,E2 -8712.639} C_VEL
LIN {X 0,Y 449.984,Z 298.268,A -85,B 0,C 180,E1 -8714.079,E2 -8714.079} C_VEL
LIN {X 0,Y 449.549,Z 311.201,A -85,B 0,C 180,E1 -8714.471,E2 -8714.471} C_VEL
LIN {X 0,Y 448.933,Z 323.796,A -85,B 0,C 180,E1 -8715.03,E2 -8715.03} C_VEL
LIN {X 0,Y 448.387,Z 335.045,A -85,B 0,C 180,E1 -8715.707,E2 -8715.707} C_VEL
LIN {X 0,Y 447.839,Z 345.99,A -85,B 0,C 180,E1 -8716.55,E2 -8716.55} C_VEL
LIN {X 0,Y 447.153,Z 357.254,A -85,B 0,C 180,E1 -8717.634,E2 -8717.634} C_VEL
LIN {X 0,Y 446.738,Z 365.883,A -85,B 0,C 180,E1 -8718.658,E2 -8718.658} C_VEL
LIN {X 0,Y 446.232,Z 373.846,A -85,B 0,C 180,E1 -8719.794,E2 -8719.794} C_VEL
LIN {X 0,Y 445.841,Z 381.631,A -85,B 0,C 180,E1 -8721.158,E2 -8721.158} C_VEL
LIN {X 0,Y 445.598,Z 388.818,A -85,B 0,C 180,E1 -8722.751,E2 -8722.751} C_VEL
LIN {X 0,Y 445.442,Z 393.208,A -85,B 0,C 180,E1 -8723.99,E2 -8723.99} C_VEL
LIN {X 0,Y 445.412,Z 397.264,A -85,B 0,C 180,E1 -8725.475,E2 -8725.475} C_VEL
LIN {X 0,Y 445.393,Z 399.151,A -85,B 0,C 180,E1 -8726.381,E2 -8726.381} C_VEL
LIN {X 0,Y 445.451,Z 400.571,A -85,B 0,C 180,E1 -8727.287,E2 -8727.287} C_VEL
LIN {X 0,Y 445.401,Z 402.205,A -85,B 0,C 180,E1 -8729.095,E2 -8729.095} C_VEL
LIN {X 0,Y 445.41,Z 402.419,A -85,B 0,C 180,E1 -8729.999,E2 -8729.999} C_VEL
LIN {X 0,Y 445.401,Z 402.196,A -85,B 0,C 180,E1 -8730.904,E2 -8730.904} C_VEL
LIN {X 0,Y 445.451,Z 400.571,A -85,B 0,C 180,E1 -8732.712,E2 -8732.712} C_VEL
LIN {X 0,Y 445.394,Z 399.136,A -85,B 0,C 180,E1 -8733.618,E2 -8733.618} C_VEL
LIN {X 0,Y 445.468,Z 396.15,A -85,B 0,C 180,E1 -8734.977,E2 -8734.977} C_VEL
LIN {X 0,Y 445.491,Z 392.097,A -85,B 0,C 180,E1 -8736.34,E2 -8736.34} C_VEL
LIN {X 0,Y 445.699,Z 385.856,A -85,B 0,C 180,E1 -8737.93,E2 -8737.93} C_VEL
LIN {X 0,Y 445.975,Z 379.049,A -85,B 0,C 180,E1 -8739.295,E2 -8739.295} C_VEL
LIN {X 0,Y 446.366,Z 370.59,A -85,B 0,C 180,E1 -8740.661,E2 -8740.661} C_VEL
LIN {X 0,Y 446.889,Z 361.872,A -85,B 0,C 180,E1 -8741.796,E2 -8741.796} C_VEL
LIN {X 0,Y 447.398,Z 352.044,A -85,B 0,C 180,E1 -8742.846,E2 -8742.846} C_VEL
LIN {X 0,Y 447.932,Z 341.905,A -85,B 0,C 180,E1 -8743.727,E2 -8743.727} C_VEL
LIN {X 0,Y 448.519,Z 330.503,A -85,B 0,C 180,E1 -8744.519,E2 -8744.519} C_VEL
LIN {X 0,Y 449.028,Z 318.814,A -85,B 0,C 180,E1 -8745.14,E2 -8745.14} C_VEL
LIN {X 0,Y 449.543,Z 305.407,A -85,B 0,C 180,E1 -8745.645,E2 -8745.645} C_VEL
LIN {X 0,Y 449.834,Z 292.283,A -85,B 0,C 180,E1 -8745.954,E2 -8745.954} C_VEL
LIN {X 0,Y 450.531,Z 211.593,A -85,B 0,C 180,E1 -8747.285,E2 -8747.285} C_VEL
LIN {X 0,Y 447.297,Z 189.501,A -85,B 0,C 180,E1 -8747.794,E2 -8747.794} C_VEL
LIN {X 0,Y 448.04,Z 173.142,A -85,B 0,C 180,E1 -8750.667,E2 -8750.667} C_VEL
LIN {X 0,Y 449.108,Z 154.304,A -85,B 0,C 180,E1 -8754.008,E2 -8754.008} C_VEL
LIN {X 0,Y 448.937,Z 150.15,A -85,B 0,C 180,E1 -8754.772,E2 -8754.772} C_VEL
LIN {X 0,Y 446.512,Z 137.867,A -85,B 0,C 180,E1 -8757.19,E2 -8757.19} C_VEL
LIN {X 0,Y 446.428,Z 137.878,A -85,B 0,C 180,E1 -8760.249,E2 -8760.249} C_VEL
LIN {X 0,Y 446.446,Z 137.871,A -85,B 0,C 180,E1 -8763.453,E2 -8763.453} C_VEL
LIN {X 0,Y 446.402,Z 137.875,A -85,B 0,C 180,E1 -8766.745,E2 -8766.745} C_VEL
LIN {X 0,Y 446.478,Z 137.869,A -85,B 0,C 180,E1 -8769.528,E2 -8769.528} C_VEL
LIN {X 0,Y 446.428,Z 137.872,A -85,B 0,C 180,E1 -8772.604,E2 -8772.604} C_VEL
LIN {X 0,Y 446.451,Z 137.87,A -85,B 0,C 180,E1 -8775.103,E2 -8775.103} C_VEL
LIN {X 0,Y 446.428,Z 137.872,A -85,B 0,C 180,E1 -8778.608,E2 -8778.608} C_VEL
LIN {X 0,Y 446.437,Z 137.871,A -85,B 0,C 180,E1 -8780.972,E2 -8780.972} C_VEL
LIN {X 0,Y 446.417,Z 137.873,A -85,B 0,C 180,E1 -8784.373,E2 -8784.373} C_VEL
LIN {X 0,Y 446.419,Z 137.879,A -85,B 0,C 180,E1 -8787.638,E2 -8787.638} C_VEL
LIN {X 0,Y 446.447,Z 137.87,A -85,B 0,C 180,E1 -8790.79,E2 -8790.79} C_VEL
LIN {X 0,Y 446.477,Z 137.868,A -85,B 0,C 180,E1 -8793.848,E2 -8793.848} C_VEL
LIN {X 0,Y 446.428,Z 137.874,A -85,B 0,C 180,E1 -8796.823,E2 -8796.823} C_VEL
LIN {X 0,Y 446.443,Z 137.872,A -85,B 0,C 180,E1 -8799.737,E2 -8799.737} C_VEL
LIN {X 0,Y 446.455,Z 137.869,A -85,B 0,C 180,E1 -8802.596,E2 -8802.596} C_VEL
LIN {X 0,Y 446.469,Z 137.871,A -85,B 0,C 180,E1 -8805.412,E2 -8805.412} C_VEL
LIN {X 0,Y 446.516,Z 137.861,A -85,B 0,C 180,E1 -8808.193,E2 -8808.193} C_VEL
LIN {X 0,Y 446.599,Z 137.851,A -85,B 0,C 180,E1 -8811.857,E2 -8811.857} C_VEL
LIN {X 0,Y 446.64,Z 137.848,A -85,B 0,C 180,E1 -8814.582,E2 -8814.582} C_VEL
LIN {X 0,Y 446.707,Z 137.84,A -85,B 0,C 180,E1 -8817.294,E2 -8817.294} C_VEL
LIN {X 0,Y 446.792,Z 137.826,A -85,B 0,C 180,E1 -8820,E2 -8820} C_VEL
LIN {X 0,Y 446.706,Z 137.844,A -85,B 0,C 180,E1 -8822.705,E2 -8822.705} C_VEL
LIN {X 0,Y 446.637,Z 137.849,A -85,B 0,C 180,E1 -8826.323,E2 -8826.323} C_VEL
LIN {X 0,Y 446.536,Z 137.861,A -85,B 0,C 180,E1 -8829.055,E2 -8829.055} C_VEL
LIN {X 0,Y 446.518,Z 137.866,A -85,B 0,C 180,E1 -8832.729,E2 -8832.729} C_VEL
LIN {X 0,Y 446.493,Z 137.868,A -85,B 0,C 180,E1 -8836.228,E2 -8836.228} C_VEL
LIN {X 0,Y 446.466,Z 137.867,A -85,B 0,C 180,E1 -8839.303,E2 -8839.303} C_VEL
LIN {X 0,Y 446.415,Z 137.879,A -85,B 0,C 180,E1 -8842.199,E2 -8842.199} C_VEL
LIN {X 0,Y 446.454,Z 137.869,A -85,B 0,C 180,E1 -8845.152,E2 -8845.152} C_VEL
LIN {X 0,Y 446.48,Z 137.872,A -85,B 0,C 180,E1 -8848.178,E2 -8848.178} C_VEL
LIN {X 0,Y 446.416,Z 137.876,A -85,B 0,C 180,E1 -8851.775,E2 -8851.775} C_VEL
LIN {X 0,Y 446.426,Z 137.875,A -85,B 0,C 180,E1 -8854.523,E2 -8854.523} C_VEL
LIN {X 0,Y 446.434,Z 137.879,A -85,B 0,C 180,E1 -8858.083,E2 -8858.083} C_VEL
LIN {X 0,Y 446.442,Z 137.87,A -85,B 0,C 180,E1 -8860.921,E2 -8860.921} C_VEL
LIN {X 0,Y 446.44,Z 137.877,A -85,B 0,C 180,E1 -8863.84,E2 -8863.84} C_VEL
LIN {X 0,Y 446.442,Z 137.872,A -85,B 0,C 180,E1 -8866.397,E2 -8866.397} C_VEL
LIN {X 0,Y 446.464,Z 137.875,A -85,B 0,C 180,E1 -8869.805,E2 -8869.805} C_VEL
LIN {X 0,Y 446.429,Z 137.875,A -85,B 0,C 180,E1 -8872.124,E2 -8872.124} C_VEL
LIN {X 0,Y 446.425,Z 137.877,A -85,B 0,C 180,E1 -8875.477,E2 -8875.477} C_VEL
LIN {X 0,Y 446.411,Z 137.874,A -85,B 0,C 180,E1 -8878.7,E2 -8878.7} C_VEL
LIN {X 0,Y 446.479,Z 137.87,A -85,B 0,C 180,E1 -8881.822,E2 -8881.822} C_VEL
LIN {X 0,Y 446.453,Z 137.869,A -85,B 0,C 180,E1 -8884.848,E2 -8884.848} C_VEL
LIN {X 0,Y 446.443,Z 137.87,A -85,B 0,C 180,E1 -8888.245,E2 -8888.245} C_VEL
LIN {X 0,Y 446.453,Z 137.873,A -85,B 0,C 180,E1 -8891.65,E2 -8891.65} C_VEL
LIN {X 0,Y 446.504,Z 137.862,A -85,B 0,C 180,E1 -8894.48,E2 -8894.48} C_VEL
LIN {X 0,Y 446.514,Z 137.861,A -85,B 0,C 180,E1 -8898.193,E2 -8898.193} C_VEL
LIN {X 0,Y 446.596,Z 137.851,A -85,B 0,C 180,E1 -8901.858,E2 -8901.858} C_VEL
LIN {X 0,Y 446.644,Z 137.846,A -85,B 0,C 180,E1 -8904.583,E2 -8904.583} C_VEL
LIN {X 0,Y 446.619,Z 137.85,A -85,B 0,C 180,E1 -8907.003,E2 -8907.003} C_VEL
LIN {X 0,Y 446.102,Z 137.92,A -85,B 0,C 180,E1 -8907.756,E2 -8907.756} C_VEL
LIN {X 0,Y 443.287,Z 138.278,A -85,B 0,C 180,E1 -8908.979,E2 -8908.979} C_VEL
LIN {X 0,Y 440.802,Z 138.588,A -85,B 0,C 180,E1 -8909.966,E2 -8909.966} C_VEL
LIN {X 0,Y 439.713,Z 138.717,A -85,B 0,C 180,E1 -8910.729,E2 -8910.729} C_VEL
LIN {X 0,Y 439.619,Z 138.726,A -85,B 0,C 180,E1 -8910.988,E2 -8910.988} C_VEL
LIN {X 0,Y 439.653,Z 138.721,A -85,B 0,C 180,E1 -8912.749,E2 -8912.749} C_VEL
LIN {X 0,Y 439.617,Z 138.723,A -85,B 0,C 180,E1 -8916.426,E2 -8916.426} C_VEL
LIN {X 0,Y 439.497,Z 138.738,A -85,B 0,C 180,E1 -8919.202,E2 -8919.202} C_VEL
LIN {X 0,Y 439.463,Z 138.745,A -85,B 0,C 180,E1 -8922.938,E2 -8922.938} C_VEL
LIN {X 0,Y 439.478,Z 138.744,A -85,B 0,C 180,E1 -8926.364,E2 -8926.364} C_VEL
LIN {X 0,Y 439.49,Z 138.926,A -85,B 0,C 180,E1 -8927.208,E2 -8927.208} C_VEL
LIN {X 0,Y 440.784,Z 147.062,A -85,B 0,C 180,E1 -8929.079,E2 -8929.079} C_VEL
LIN {X 0,Y 440.733,Z 151.361,A -85,B 0,C 180,E1 -8930.023,E2 -8930.023} C_VEL
LIN {X 0,Y 444.158,Z 168.598,A -85,B 0,C 180,E1 -8930.468,E2 -8930.468} C_VEL
LIN {X 0,Y 443.042,Z 258.202,A -85,B 0,C 180,E1 -8931.98,E2 -8931.98} C_VEL
LIN {X 0,Y 442.697,Z 271.849,A -85,B 0,C 180,E1 -8932.397,E2 -8932.397} C_VEL
LIN {X 0,Y 442.357,Z 284.453,A -85,B 0,C 180,E1 -8932.974,E2 -8932.974} C_VEL
LIN {X 0,Y 441.958,Z 295.805,A -85,B 0,C 180,E1 -8933.674,E2 -8933.674} C_VEL
LIN {X 0,Y 441.324,Z 307.145,A -85,B 0,C 180,E1 -8934.569,E2 -8934.569} C_VEL
LIN {X 0,Y 440.715,Z 317.86,A -85,B 0,C 180,E1 -8935.631,E2 -8935.631} C_VEL
LIN {X 0,Y 440.209,Z 327.231,A -85,B 0,C 180,E1 -8936.784,E2 -8936.784} C_VEL
LIN {X 0,Y 439.677,Z 336.048,A -85,B 0,C 180,E1 -8938.129,E2 -8938.129} C_VEL
LIN {X 0,Y 439.257,Z 343.176,A -85,B 0,C 180,E1 -8939.472,E2 -8939.472} C_VEL
LIN {X 0,Y 438.923,Z 348.947,A -85,B 0,C 180,E1 -8940.823,E2 -8940.823} C_VEL
LIN {X 0,Y 438.615,Z 354.367,A -85,B 0,C 180,E1 -8942.465,E2 -8942.465} C_VEL
LIN {X 0,Y 438.423,Z 358.296,A -85,B 0,C 180,E1 -8944.13,E2 -8944.13} C_VEL
LIN {X 0,Y 438.293,Z 360.169,A -85,B 0,C 180,E1 -8945.259,E2 -8945.259} C_VEL
LIN {X 0,Y 438.24,Z 361.635,A -85,B 0,C 180,E1 -8946.694,E2 -8946.694} C_VEL
LIN {X 0,Y 438.225,Z 362.116,A -85,B 0,C 180,E1 -8948.203,E2 -8948.203} C_VEL
LIN {X 0,Y 438.244,Z 361.366,A -85,B 0,C 180,E1 -8949.902,E2 -8949.902} C_VEL
LIN {X 0,Y 438.415,Z 359.104,A -85,B 0,C 180,E1 -8951.703,E2 -8951.703} C_VEL
LIN {X 0,Y 438.598,Z 356.463,A -85,B 0,C 180,E1 -8952.991,E2 -8952.991} C_VEL
LIN {X 0,Y 438.78,Z 352.883,A -85,B 0,C 180,E1 -8954.299,E2 -8954.299} C_VEL
LIN {X 0,Y 439.008,Z 348.303,A -85,B 0,C 180,E1 -8955.608,E2 -8955.608} C_VEL
LIN {X 0,Y 439.446,Z 341.55,A -85,B 0,C 180,E1 -8957.131,E2 -8957.131} C_VEL
LIN {X 0,Y 439.955,Z 333.833,A -85,B 0,C 180,E1 -8958.503,E2 -8958.503} C_VEL
LIN {X 0,Y 440.532,Z 324.679,A -85,B 0,C 180,E1 -8959.815,E2 -8959.815} C_VEL
LIN {X 0,Y 441.142,Z 315.459,A -85,B 0,C 180,E1 -8960.888,E2 -8960.888} C_VEL
LIN {X 0,Y 441.718,Z 304.765,A -85,B 0,C 180,E1 -8961.897,E2 -8961.897} C_VEL
LIN {X 0,Y 442.403,Z 292.672,A -85,B 0,C 180,E1 -8962.789,E2 -8962.789} C_VEL
LIN {X 0,Y 442.913,Z 280.402,A -85,B 0,C 180,E1 -8963.482,E2 -8963.482} C_VEL
LIN {X 0,Y 443.225,Z 267.317,A -85,B 0,C 180,E1 -8964.007,E2 -8964.007} C_VEL
LIN {X 0,Y 443.508,Z 254.481,A -85,B 0,C 180,E1 -8964.332,E2 -8964.332} C_VEL
LIN {X 0,Y 444.459,Z 167.95,A -85,B 0,C 180,E1 -8965.806,E2 -8965.806} C_VEL
LIN {X 0,Y 441.016,Z 151.96,A -85,B 0,C 180,E1 -8966.272,E2 -8966.272} C_VEL
LIN {X 0,Y 440.852,Z 146.124,A -85,B 0,C 180,E1 -8967.528,E2 -8967.528} C_VEL
LIN {X 0,Y 439.399,Z 138.754,A -85,B 0,C 180,E1 -8969.215,E2 -8969.215} C_VEL
LIN {X 0,Y 439.439,Z 138.747,A -85,B 0,C 180,E1 -8972.368,E2 -8972.368} C_VEL
LIN {X 0,Y 439.411,Z 138.752,A -85,B 0,C 180,E1 -8975.738,E2 -8975.738} C_VEL
LIN {X 0,Y 439.391,Z 138.754,A -85,B 0,C 180,E1 -8979.398,E2 -8979.398} C_VEL
LIN {X 0,Y 439.407,Z 138.75,A -85,B 0,C 180,E1 -8982.309,E2 -8982.309} C_VEL
LIN {X 0,Y 439.449,Z 138.748,A -85,B 0,C 180,E1 -8985.175,E2 -8985.175} C_VEL
LIN {X 0,Y 439.487,Z 138.741,A -85,B 0,C 180,E1 -8988.002,E2 -8988.002} C_VEL
LIN {X 0,Y 439.508,Z 138.738,A -85,B 0,C 180,E1 -8991.726,E2 -8991.726} C_VEL
LIN {X 0,Y 439.602,Z 138.729,A -85,B 0,C 180,E1 -8994.496,E2 -8994.496} C_VEL
LIN {X 0,Y 439.632,Z 138.725,A -85,B 0,C 180,E1 -8998.168,E2 -8998.168} C_VEL
LIN {X 0,Y 439.673,Z 138.714,A -85,B 0,C 180,E1 -9000.001,E2 -9000.001} C_VEL
LIN {X 0,Y 439.607,Z 138.719,A -85,B 0,C 180,E1 -9002.75,E2 -9002.75} C_VEL
LIN {X 0,Y 439.562,Z 138.724,A -85,B 0,C 180,E1 -9006.427,E2 -9006.427} C_VEL
LIN {X 0,Y 439.477,Z 138.739,A -85,B 0,C 180,E1 -9009.203,E2 -9009.203} C_VEL
LIN {X 0,Y 439.456,Z 138.741,A -85,B 0,C 180,E1 -9012.938,E2 -9012.938} C_VEL
LIN {X 0,Y 439.4,Z 138.748,A -85,B 0,C 180,E1 -9016.325,E2 -9016.325} C_VEL
LIN {X 0,Y 439.36,Z 138.753,A -85,B 0,C 180,E1 -9019.629,E2 -9019.629} C_VEL
LIN {X 0,Y 439.354,Z 138.754,A -85,B 0,C 180,E1 -9022.577,E2 -9022.577} C_VEL
LIN {X 0,Y 439.355,Z 138.758,A -85,B 0,C 180,E1 -9025.588,E2 -9025.588} C_VEL
LIN {X 0,Y 439.381,Z 138.749,A -85,B 0,C 180,E1 -9028.677,E2 -9028.677} C_VEL
LIN {X 0,Y 439.357,Z 138.751,A -85,B 0,C 180,E1 -9032.026,E2 -9032.026} C_VEL
LIN {X 0,Y 439.396,Z 138.751,A -85,B 0,C 180,E1 -9035.339,E2 -9035.339} C_VEL
LIN {X 0,Y 439.367,Z 138.754,A -85,B 0,C 180,E1 -9038.597,E2 -9038.597} C_VEL
LIN {X 0,Y 439.353,Z 138.756,A -85,B 0,C 180,E1 -9042.21,E2 -9042.21} C_VEL
LIN {X 0,Y 439.403,Z 138.752,A -85,B 0,C 180,E1 -9045.27,E2 -9045.27} C_VEL
LIN {X 0,Y 439.362,Z 138.757,A -85,B 0,C 180,E1 -9049.016,E2 -9049.016} C_VEL
LIN {X 0,Y 439.369,Z 138.755,A -85,B 0,C 180,E1 -9051.609,E2 -9051.609} C_VEL
LIN {X 0,Y 439.403,Z 138.751,A -85,B 0,C 180,E1 -9054.844,E2 -9054.844} C_VEL
LIN {X 0,Y 439.378,Z 138.762,A -85,B 0,C 180,E1 -9058.139,E2 -9058.139} C_VEL
LIN {X 0,Y 439.414,Z 138.752,A -85,B 0,C 180,E1 -9061.604,E2 -9061.604} C_VEL
LIN {X 0,Y 439.421,Z 138.798,A -85,B 0,C 180,E1 -9062.656,E2 -9062.656} C_VEL
LIN {X 0,Y 441.887,Z 150.754,A -85,B 0,C 180,E1 -9065.035,E2 -9065.035} C_VEL
LIN {X 0,Y 442.13,Z 155.04,A -85,B 0,C 180,E1 -9065.838,E2 -9065.838} C_VEL
LIN {X 0,Y 441.107,Z 172.663,A -85,B 0,C 180,E1 -9068.992,E2 -9068.992} C_VEL
LIN {X 0,Y 440.418,Z 188.281,A -85,B 0,C 180,E1 -9071.757,E2 -9071.757} C_VEL
LIN {X 0,Y 444.048,Z 212.528,A -85,B 0,C 180,E1 -9072.344,E2 -9072.344} C_VEL
LIN {X 0,Y 443.198,Z 297.234,A -85,B 0,C 180,E1 -9073.799,E2 -9073.799} C_VEL
LIN {X 0,Y 442.707,Z 310.371,A -85,B 0,C 180,E1 -9074.195,E2 -9074.195} C_VEL
LIN {X 0,Y 442.081,Z 323.635,A -85,B 0,C 180,E1 -9074.792,E2 -9074.792} C_VEL
LIN {X 0,Y 441.5,Z 334.832,A -85,B 0,C 180,E1 -9075.48,E2 -9075.48} C_VEL
LIN {X 0,Y 440.886,Z 346.21,A -85,B 0,C 180,E1 -9076.375,E2 -9076.375} C_VEL
LIN {X 0,Y 440.169,Z 357.004,A -85,B 0,C 180,E1 -9077.435,E2 -9077.435} C_VEL
LIN {X 0,Y 439.735,Z 365.616,A -85,B 0,C 180,E1 -9078.475,E2 -9078.475} C_VEL
LIN {X 0,Y 439.188,Z 373.564,A -85,B 0,C 180,E1 -9079.628,E2 -9079.628} C_VEL
LIN {X 0,Y 438.788,Z 381.337,A -85,B 0,C 180,E1 -9081.015,E2 -9081.015} C_VEL
LIN {X 0,Y 438.524,Z 388.518,A -85,B 0,C 180,E1 -9082.633,E2 -9082.633} C_VEL
LIN {X 0,Y 438.343,Z 393.34,A -85,B 0,C 180,E1 -9084.031,E2 -9084.031} C_VEL
LIN {X 0,Y 438.341,Z 396.957,A -85,B 0,C 180,E1 -9085.401,E2 -9085.401} C_VEL
LIN {X 0,Y 438.294,Z 398.839,A -85,B 0,C 180,E1 -9086.322,E2 -9086.322} C_VEL
LIN {X 0,Y 438.376,Z 400.256,A -85,B 0,C 180,E1 -9087.243,E2 -9087.243} C_VEL
LIN {X 0,Y 438.311,Z 401.885,A -85,B 0,C 180,E1 -9089.081,E2 -9089.081} C_VEL
LIN {X 0,Y 438.318,Z 402.094,A -85,B 0,C 180,E1 -9089.999,E2 -9089.999} C_VEL
LIN {X 0,Y 438.311,Z 401.866,A -85,B 0,C 180,E1 -9090.918,E2 -9090.918} C_VEL
LIN {X 0,Y 438.376,Z 400.235,A -85,B 0,C 180,E1 -9092.756,E2 -9092.756} C_VEL
LIN {X 0,Y 438.296,Z 398.789,A -85,B 0,C 180,E1 -9093.677,E2 -9093.677} C_VEL
LIN {X 0,Y 438.376,Z 395.795,A -85,B 0,C 180,E1 -9095.058,E2 -9095.058} C_VEL
LIN {X 0,Y 438.425,Z 391.73,A -85,B 0,C 180,E1 -9096.442,E2 -9096.442} C_VEL
LIN {X 0,Y 438.65,Z 385.471,A -85,B 0,C 180,E1 -9098.058,E2 -9098.058} C_VEL
LIN {X 0,Y 438.928,Z 378.646,A -85,B 0,C 180,E1 -9099.446,E2 -9099.446} C_VEL
LIN {X 0,Y 439.355,Z 370.161,A -85,B 0,C 180,E1 -9100.833,E2 -9100.833} C_VEL
LIN {X 0,Y 439.888,Z 361.416,A -85,B 0,C 180,E1 -9101.987,E2 -9101.987} C_VEL
LIN {X 0,Y 440.448,Z 351.13,A -85,B 0,C 180,E1 -9103.095,E2 -9103.095} C_VEL
LIN {X 0,Y 441.093,Z 339.947,A -85,B 0,C 180,E1 -9104.062,E2 -9104.062} C_VEL
LIN {X 0,Y 441.728,Z 327.973,A -85,B 0,C 180,E1 -9104.865,E2 -9104.865} C_VEL
LIN {X 0,Y 442.324,Z 315.534,A -85,B 0,C 180,E1 -9105.493,E2 -9105.493} C_VEL
LIN {X 0,Y 442.771,Z 302.713,A -85,B 0,C 180,E1 -9105.949,E2 -9105.949} C_VEL
LIN {X 0,Y 443.074,Z 287.521,A -85,B 0,C 180,E1 -9106.263,E2 -9106.263} C_VEL
LIN {X 0,Y 443.79,Z 213.094,A -85,B 0,C 180,E1 -9107.511,E2 -9107.511} C_VEL
LIN {X 0,Y 440.35,Z 189.123,A -85,B 0,C 180,E1 -9108.084,E2 -9108.084} C_VEL
LIN {X 0,Y 441.057,Z 174.091,A -85,B 0,C 180,E1 -9110.765,E2 -9110.765} C_VEL
LIN {X 0,Y 442.174,Z 155.266,A -85,B 0,C 180,E1 -9114.159,E2 -9114.159} C_VEL
LIN {X 0,Y 441.901,Z 150.964,A -85,B 0,C 180,E1 -9114.969,E2 -9114.969} C_VEL
LIN {X 0,Y 439.464,Z 138.745,A -85,B 0,C 180,E1 -9117.404,E2 -9117.404} C_VEL
LIN {X 0,Y 439.362,Z 138.753,A -85,B 0,C 180,E1 -9120.788,E2 -9120.788} C_VEL
LIN {X 0,Y 439.388,Z 138.756,A -85,B 0,C 180,E1 -9124.043,E2 -9124.043} C_VEL
LIN {X 0,Y 439.349,Z 138.753,A -85,B 0,C 180,E1 -9126.886,E2 -9126.886} C_VEL
LIN {X 0,Y 439.414,Z 138.753,A -85,B 0,C 180,E1 -9129.85,E2 -9129.85} C_VEL
LIN {X 0,Y 439.381,Z 138.75,A -85,B 0,C 180,E1 -9132.626,E2 -9132.626} C_VEL
LIN {X 0,Y 439.399,Z 138.749,A -85,B 0,C 180,E1 -9135.27,E2 -9135.27} C_VEL
LIN {X 0,Y 439.388,Z 138.749,A -85,B 0,C 180,E1 -9138.743,E2 -9138.743} C_VEL
LIN {X 0,Y 439.371,Z 138.758,A -85,B 0,C 180,E1 -9141.608,E2 -9141.608} C_VEL
LIN {X 0,Y 439.395,Z 138.748,A -85,B 0,C 180,E1 -9144.843,E2 -9144.843} C_VEL
LIN {X 0,Y 439.37,Z 138.752,A -85,B 0,C 180,E1 -9148.139,E2 -9148.139} C_VEL
LIN {X 0,Y 439.431,Z 138.749,A -85,B 0,C 180,E1 -9151.598,E2 -9151.598} C_VEL
LIN {X 0,Y 439.404,Z 138.747,A -85,B 0,C 180,E1 -9154.415,E2 -9154.415} C_VEL
LIN {X 0,Y 439.364,Z 138.758,A -85,B 0,C 180,E1 -9157.424,E2 -9157.424} C_VEL
LIN {X 0,Y 439.439,Z 138.744,A -85,B 0,C 180,E1 -9160.663,E2 -9160.663} C_VEL
LIN {X 0,Y 439.461,Z 138.74,A -85,B 0,C 180,E1 -9164.224,E2 -9164.224} C_VEL
LIN {X 0,Y 439.482,Z 138.737,A -85,B 0,C 180,E1 -9168.001,E2 -9168.001} C_VEL
LIN {X 0,Y 439.546,Z 138.73,A -85,B 0,C 180,E1 -9171.726,E2 -9171.726} C_VEL
LIN {X 0,Y 439.616,Z 138.723,A -85,B 0,C 180,E1 -9174.495,E2 -9174.495} C_VEL
LIN {X 0,Y 439.635,Z 138.719,A -85,B 0,C 180,E1 -9178.167,E2 -9178.167} C_VEL
LIN {X 0,Y 439.762,Z 138.702,A -85,B 0,C 180,E1 -9179.999,E2 -9179.999} C_VEL
LIN {X 0,Y 439.653,Z 138.723,A -85,B 0,C 180,E1 -9182.748,E2 -9182.748} C_VEL
LIN {X 0,Y 439.609,Z 138.725,A -85,B 0,C 180,E1 -9186.425,E2 -9186.425} C_VEL
LIN {X 0,Y 439.498,Z 138.737,A -85,B 0,C 180,E1 -9189.201,E2 -9189.201} C_VEL
LIN {X 0,Y 439.463,Z 138.743,A -85,B 0,C 180,E1 -9192.937,E2 -9192.937} C_VEL
LIN {X 0,Y 439.444,Z 138.747,A -85,B 0,C 180,E1 -9196.348,E2 -9196.348} C_VEL
LIN {X 0,Y 439.399,Z 138.747,A -85,B 0,C 180,E1 -9199.626,E2 -9199.626} C_VEL
LIN {X 0,Y 439.361,Z 138.757,A -85,B 0,C 180,E1 -9202.575,E2 -9202.575} C_VEL
LIN {X 0,Y 439.401,Z 138.748,A -85,B 0,C 180,E1 -9205.584,E2 -9205.584} C_VEL
LIN {X 0,Y 439.413,Z 138.748,A -85,B 0,C 180,E1 -9208.673,E2 -9208.673} C_VEL
LIN {X 0,Y 439.367,Z 138.757,A -85,B 0,C 180,E1 -9212.03,E2 -9212.03} C_VEL
LIN {X 0,Y 439.391,Z 138.749,A -85,B 0,C 180,E1 -9215.341,E2 -9215.341} C_VEL
LIN {X 0,Y 439.394,Z 138.749,A -85,B 0,C 180,E1 -9218.593,E2 -9218.593} C_VEL
LIN {X 0,Y 439.4,Z 138.748,A -85,B 0,C 180,E1 -9221.259,E2 -9221.259} C_VEL
LIN {X 0,Y 439.405,Z 138.747,A -85,B 0,C 180,E1 -9224.728,E2 -9224.728} C_VEL
LIN {X 0,Y 439.407,Z 138.753,A -85,B 0,C 180,E1 -9227.798,E2 -9227.798} C_VEL
LIN {X 0,Y 439.447,Z 138.744,A -85,B 0,C 180,E1 -9230.23,E2 -9230.23} C_VEL
LIN {X 0,Y 439.372,Z 138.758,A -85,B 0,C 180,E1 -9233.713,E2 -9233.713} C_VEL
LIN {X 0,Y 439.367,Z 138.752,A -85,B 0,C 180,E1 -9237.054,E2 -9237.054} C_VEL
LIN {X 0,Y 439.377,Z 138.751,A -85,B 0,C 180,E1 -9240.274,E2 -9240.274} C_VEL
LIN {X 0,Y 439.425,Z 138.75,A -85,B 0,C 180,E1 -9243.397,E2 -9243.397} C_VEL
LIN {X 0,Y 439.382,Z 138.749,A -85,B 0,C 180,E1 -9246.43,E2 -9246.43} C_VEL
LIN {X 0,Y 439.385,Z 138.757,A -85,B 0,C 180,E1 -9249.397,E2 -9249.397} C_VEL
LIN {X 0,Y 439.427,Z 138.744,A -85,B 0,C 180,E1 -9252.31,E2 -9252.31} C_VEL
LIN {X 0,Y 439.445,Z 138.748,A -85,B 0,C 180,E1 -9255.174,E2 -9255.174} C_VEL
LIN {X 0,Y 439.48,Z 138.738,A -85,B 0,C 180,E1 -9258.002,E2 -9258.002} C_VEL
LIN {X 0,Y 439.544,Z 138.731,A -85,B 0,C 180,E1 -9261.727,E2 -9261.727} C_VEL
LIN {X 0,Y 439.619,Z 138.721,A -85,B 0,C 180,E1 -9264.496,E2 -9264.496} C_VEL
LIN {X 0,Y 439.632,Z 138.718,A -85,B 0,C 180,E1 -9268.168,E2 -9268.168} C_VEL
LIN {X 0,Y 439.761,Z 138.702,A -85,B 0,C 180,E1 -9270.001,E2 -9270.001} C_VEL
LIN {X 0,Y 439.619,Z 138.726,A -85,B 0,C 180,E1 -9270.988,E2 -9270.988} C_VEL
LIN {X 0,Y 438.902,Z 138.811,A -85,B 0,C 180,E1 -9271.752,E2 -9271.752} C_VEL
LIN {X 0,Y 435.923,Z 139.187,A -85,B 0,C 180,E1 -9272.991,E2 -9272.991} C_VEL
LIN {X 0,Y 433.472,Z 139.492,A -85,B 0,C 180,E1 -9273.991,E2 -9273.991} C_VEL
LIN {X 0,Y 432.499,Z 139.613,A -85,B 0,C 180,E1 -9274.766,E2 -9274.766} C_VEL
LIN {X 0,Y 432.462,Z 139.613,A -85,B 0,C 180,E1 -9275.028,E2 -9275.028} C_VEL
LIN {X 0,Y 432.583,Z 139.597,A -85,B 0,C 180,E1 -9277.68,E2 -9277.68} C_VEL
LIN {X 0,Y 432.391,Z 139.624,A -85,B 0,C 180,E1 -9281.248,E2 -9281.248} C_VEL
LIN {X 0,Y 432.372,Z 139.627,A -85,B 0,C 180,E1 -9284.113,E2 -9284.113} C_VEL
LIN {X 0,Y 432.433,Z 139.765,A -85,B 0,C 180,E1 -9287.011,E2 -9287.011} C_VEL
LIN {X 0,Y 433.791,Z 147.904,A -85,B 0,C 180,E1 -9288.907,E2 -9288.907} C_VEL
LIN {X 0,Y 433.801,Z 151.635,A -85,B 0,C 180,E1 -9289.737,E2 -9289.737} C_VEL
LIN {X 0,Y 437.327,Z 169.063,A -85,B 0,C 180,E1 -9290.203,E2 -9290.203} C_VEL
LIN {X 0,Y 436.188,Z 259.554,A -85,B 0,C 180,E1 -9291.768,E2 -9291.768} C_VEL
LIN {X 0,Y 435.83,Z 273.245,A -85,B 0,C 180,E1 -9292.207,E2 -9292.207} C_VEL
LIN {X 0,Y 435.464,Z 285.491,A -85,B 0,C 180,E1 -9292.79,E2 -9292.79} C_VEL
LIN {X 0,Y 435.048,Z 296.519,A -85,B 0,C 180,E1 -9293.491,E2 -9293.491} C_VEL
LIN {X 0,Y 434.392,Z 307.419,A -85,B 0,C 180,E1 -9294.367,E2 -9294.367} C_VEL
LIN {X 0,Y 433.779,Z 317.972,A -85,B 0,C 180,E1 -9295.426,E2 -9295.426} C_VEL
LIN {X 0,Y 433.217,Z 327.762,A -85,B 0,C 180,E1 -9296.651,E2 -9296.651} C_VEL
LIN {X 0,Y 432.615,Z 337.073,A -85,B 0,C 180,E1 -9298.107,E2 -9298.107} C_VEL
LIN {X 0,Y 432.199,Z 344.045,A -85,B 0,C 180,E1 -9299.466,E2 -9299.466} C_VEL
LIN {X 0,Y 431.858,Z 349.81,A -85,B 0,C 180,E1 -9300.866,E2 -9300.866} C_VEL
LIN {X 0,Y 431.533,Z 355.006,A -85,B 0,C 180,E1 -9302.51,E2 -9302.51} C_VEL
LIN {X 0,Y 431.376,Z 358.095,A -85,B 0,C 180,E1 -9303.81,E2 -9303.81} C_VEL
LIN {X 0,Y 431.185,Z 360.722,A -85,B 0,C 180,E1 -9305.417,E2 -9305.417} C_VEL
LIN {X 0,Y 431.134,Z 362.177,A -85,B 0,C 180,E1 -9307.096,E2 -9307.096} C_VEL
LIN {X 0,Y 431.119,Z 362.398,A -85,B 0,C 180,E1 -9308.512,E2 -9308.512} C_VEL
LIN {X 0,Y 431.158,Z 361.653,A -85,B 0,C 180,E1 -9309.995,E2 -9309.995} C_VEL
LIN {X 0,Y 431.362,Z 359.192,A -85,B 0,C 180,E1 -9311.913,E2 -9311.913} C_VEL
LIN {X 0,Y 431.597,Z 355.242,A -85,B 0,C 180,E1 -9313.704,E2 -9313.704} C_VEL
LIN {X 0,Y 431.889,Z 350.28,A -85,B 0,C 180,E1 -9315.306,E2 -9315.306} C_VEL
LIN {X 0,Y 432.266,Z 344.954,A -85,B 0,C 180,E1 -9316.635,E2 -9316.635} C_VEL
LIN {X 0,Y 432.701,Z 338.474,A -85,B 0,C 180,E1 -9317.948,E2 -9317.948} C_VEL
LIN {X 0,Y 433.245,Z 330.526,A -85,B 0,C 180,E1 -9319.253,E2 -9319.253} C_VEL
LIN {X 0,Y 433.885,Z 320.971,A -85,B 0,C 180,E1 -9320.524,E2 -9320.524} C_VEL
LIN {X 0,Y 434.483,Z 310.701,A -85,B 0,C 180,E1 -9321.631,E2 -9321.631} C_VEL
LIN {X 0,Y 435.188,Z 300.001,A -85,B 0,C 180,E1 -9322.545,E2 -9322.545} C_VEL
LIN {X 0,Y 435.829,Z 287.652,A -85,B 0,C 180,E1 -9323.371,E2 -9323.371} C_VEL
LIN {X 0,Y 436.235,Z 275.525,A -85,B 0,C 180,E1 -9323.983,E2 -9323.983} C_VEL
LIN {X 0,Y 436.525,Z 263.018,A -85,B 0,C 180,E1 -9324.419,E2 -9324.419} C_VEL
LIN {X 0,Y 436.809,Z 244.807,A -85,B 0,C 180,E1 -9324.783,E2 -9324.783} C_VEL
LIN {X 0,Y 437.765,Z 169.021,A -85,B 0,C 180,E1 -9326.091,E2 -9326.091} C_VEL
LIN {X 0,Y 434.128,Z 152.392,A -85,B 0,C 180,E1 -9326.57,E2 -9326.57} C_VEL
LIN {X 0,Y 433.897,Z 147.317,A -85,B 0,C 180,E1 -9327.69,E2 -9327.69} C_VEL
LIN {X 0,Y 432.368,Z 139.631,A -85,B 0,C 180,E1 -9329.486,E2 -9329.486} C_VEL
LIN {X 0,Y 432.388,Z 139.628,A -85,B 0,C 180,E1 -9332.929,E2 -9332.929} C_VEL
LIN {X 0,Y 432.369,Z 139.628,A -85,B 0,C 180,E1 -9336.024,E2 -9336.024} C_VEL
LIN {X 0,Y 432.353,Z 139.632,A -85,B 0,C 180,E1 -9339.047,E2 -9339.047} C_VEL
LIN {X 0,Y 432.363,Z 139.626,A -85,B 0,C 180,E1 -9342.011,E2 -9342.011} C_VEL
LIN {X 0,Y 432.397,Z 139.627,A -85,B 0,C 180,E1 -9344.927,E2 -9344.927} C_VEL
LIN {X 0,Y 432.463,Z 139.616,A -85,B 0,C 180,E1 -9347.804,E2 -9347.804} C_VEL
LIN {X 0,Y 432.468,Z 139.615,A -85,B 0,C 180,E1 -9351.59,E2 -9351.59} C_VEL
LIN {X 0,Y 432.576,Z 139.606,A -85,B 0,C 180,E1 -9354.406,E2 -9354.406} C_VEL
LIN {X 0,Y 432.601,Z 139.601,A -85,B 0,C 180,E1 -9358.139,E2 -9358.139} C_VEL
LIN {X 0,Y 432.625,Z 139.592,A -85,B 0,C 180,E1 -9360.001,E2 -9360.001} C_VEL
LIN {X 0,Y 432.561,Z 139.596,A -85,B 0,C 180,E1 -9362.794,E2 -9362.794} C_VEL
LIN {X 0,Y 432.574,Z 139.601,A -85,B 0,C 180,E1 -9365.595,E2 -9365.595} C_VEL
LIN {X 0,Y 432.45,Z 139.616,A -85,B 0,C 180,E1 -9368.411,E2 -9368.411} C_VEL
LIN {X 0,Y 432.452,Z 139.616,A -85,B 0,C 180,E1 -9372.197,E2 -9372.197} C_VEL
LIN {X 0,Y 432.36,Z 139.627,A -85,B 0,C 180,E1 -9376.042,E2 -9376.042} C_VEL
LIN {X 0,Y 432.328,Z 139.628,A -85,B 0,C 180,E1 -9379.461,E2 -9379.461} C_VEL
LIN {X 0,Y 432.341,Z 139.628,A -85,B 0,C 180,E1 -9382.091,E2 -9382.091} C_VEL
LIN {X 0,Y 432.317,Z 139.631,A -85,B 0,C 180,E1 -9385.004,E2 -9385.004} C_VEL
LIN {X 0,Y 432.317,Z 139.628,A -85,B 0,C 180,E1 -9388.128,E2 -9388.128} C_VEL
LIN {X 0,Y 432.309,Z 139.631,A -85,B 0,C 180,E1 -9391.348,E2 -9391.348} C_VEL
LIN {X 0,Y 432.332,Z 139.631,A -85,B 0,C 180,E1 -9394.678,E2 -9394.678} C_VEL
LIN {X 0,Y 432.334,Z 139.628,A -85,B 0,C 180,E1 -9398.151,E2 -9398.151} C_VEL
LIN {X 0,Y 432.308,Z 139.632,A -85,B 0,C 180,E1 -9401.801,E2 -9401.801} C_VEL
LIN {X 0,Y 432.338,Z 139.631,A -85,B 0,C 180,E1 -9404.347,E2 -9404.347} C_VEL
LIN {X 0,Y 432.312,Z 139.637,A -85,B 0,C 180,E1 -9407.018,E2 -9407.018} C_VEL
LIN {X 0,Y 432.313,Z 139.635,A -85,B 0,C 180,E1 -9409.825,E2 -9409.825} C_VEL
LIN {X 0,Y 432.309,Z 139.634,A -85,B 0,C 180,E1 -9413.022,E2 -9413.022} C_VEL
LIN {X 0,Y 432.364,Z 139.632,A -85,B 0,C 180,E1 -9415.996,E2 -9415.996} C_VEL
LIN {X 0,Y 432.351,Z 139.632,A -85,B 0,C 180,E1 -9419.49,E2 -9419.49} C_VEL
LIN {X 0,Y 432.383,Z 139.796,A -85,B 0,C 180,E1 -9422.403,E2 -9422.403} C_VEL
LIN {X 0,Y 434.895,Z 151.671,A -85,B 0,C 180,E1 -9424.82,E2 -9424.82} C_VEL
LIN {X 0,Y 435.245,Z 156.181,A -85,B 0,C 180,E1 -9425.684,E2 -9425.684} C_VEL
LIN {X 0,Y 434.157,Z 173.789,A -85,B 0,C 180,E1 -9428.888,E2 -9428.888} C_VEL
LIN {X 0,Y 433.489,Z 187.906,A -85,B 0,C 180,E1 -9431.432,E2 -9431.432} C_VEL
LIN {X 0,Y 437.33,Z 213.47,A -85,B 0,C 180,E1 -9432.068,E2 -9432.068} C_VEL
LIN {X 0,Y 436.409,Z 297.456,A -85,B 0,C 180,E1 -9433.54,E2 -9433.54} C_VEL
LIN {X 0,Y 435.879,Z 311.159,A -85,B 0,C 180,E1 -9433.971,E2 -9433.971} C_VEL
LIN {X 0,Y 435.238,Z 323.556,A -85,B 0,C 180,E1 -9434.547,E2 -9434.547} C_VEL
LIN {X 0,Y 434.523,Z 336.26,A -85,B 0,C 180,E1 -9435.361,E2 -9435.361} C_VEL
LIN {X 0,Y 433.85,Z 347.917,A -85,B 0,C 180,E1 -9436.325,E2 -9436.325} C_VEL
LIN {X 0,Y 433.152,Z 357.816,A -85,B 0,C 180,E1 -9437.347,E2 -9437.347} C_VEL
LIN {X 0,Y 432.646,Z 367.045,A -85,B 0,C 180,E1 -9438.521,E2 -9438.521} C_VEL
LIN {X 0,Y 432.013,Z 376.055,A -85,B 0,C 180,E1 -9439.928,E2 -9439.928} C_VEL
LIN {X 0,Y 431.649,Z 383.317,A -85,B 0,C 180,E1 -9441.337,E2 -9441.337} C_VEL
LIN {X 0,Y 431.439,Z 388.228,A -85,B 0,C 180,E1 -9442.512,E2 -9442.512} C_VEL
LIN {X 0,Y 431.244,Z 393.464,A -85,B 0,C 180,E1 -9444.072,E2 -9444.072} C_VEL
LIN {X 0,Y 431.269,Z 396.654,A -85,B 0,C 180,E1 -9445.326,E2 -9445.326} C_VEL
LIN {X 0,Y 431.199,Z 398.528,A -85,B 0,C 180,E1 -9446.261,E2 -9446.261} C_VEL
LIN {X 0,Y 431.284,Z 399.943,A -85,B 0,C 180,E1 -9447.197,E2 -9447.197} C_VEL
LIN {X 0,Y 431.243,Z 400.951,A -85,B 0,C 180,E1 -9448.132,E2 -9448.132} C_VEL
LIN {X 0,Y 431.225,Z 401.566,A -85,B 0,C 180,E1 -9449.066,E2 -9449.066} C_VEL
LIN {X 0,Y 431.229,Z 401.767,A -85,B 0,C 180,E1 -9449.999,E2 -9449.999} C_VEL
LIN {X 0,Y 431.224,Z 401.536,A -85,B 0,C 180,E1 -9450.933,E2 -9450.933} C_VEL
LIN {X 0,Y 431.242,Z 400.914,A -85,B 0,C 180,E1 -9451.867,E2 -9451.867} C_VEL
LIN {X 0,Y 431.284,Z 399.897,A -85,B 0,C 180,E1 -9452.802,E2 -9452.802} C_VEL
LIN {X 0,Y 431.201,Z 398.441,A -85,B 0,C 180,E1 -9453.737,E2 -9453.737} C_VEL
LIN {X 0,Y 431.284,Z 395.436,A -85,B 0,C 180,E1 -9455.142,E2 -9455.142} C_VEL
LIN {X 0,Y 431.342,Z 391.358,A -85,B 0,C 180,E1 -9456.548,E2 -9456.548} C_VEL
LIN {X 0,Y 431.579,Z 385.08,A -85,B 0,C 180,E1 -9458.191,E2 -9458.191} C_VEL
LIN {X 0,Y 431.876,Z 378.237,A -85,B 0,C 180,E1 -9459.601,E2 -9459.601} C_VEL
LIN {X 0,Y 432.362,Z 369.719,A -85,B 0,C 180,E1 -9461.01,E2 -9461.01} C_VEL
LIN {X 0,Y 432.898,Z 360.942,A -85,B 0,C 180,E1 -9462.183,E2 -9462.183} C_VEL
LIN {X 0,Y 433.489,Z 350.37,A -85,B 0,C 180,E1 -9463.334,E2 -9463.334} C_VEL
LIN {X 0,Y 434.147,Z 339.378,A -85,B 0,C 180,E1 -9464.292,E2 -9464.292} C_VEL
LIN {X 0,Y 434.831,Z 327.317,A -85,B 0,C 180,E1 -9465.106,E2 -9465.106} C_VEL
LIN {X 0,Y 435.4,Z 316.075,A -85,B 0,C 180,E1 -9465.686,E2 -9465.686} C_VEL
LIN {X 0,Y 435.887,Z 303.649,A -85,B 0,C 180,E1 -9466.148,E2 -9466.148} C_VEL
LIN {X 0,Y 436.152,Z 291.257,A -85,B 0,C 180,E1 -9466.439,E2 -9466.439} C_VEL
LIN {X 0,Y 436.977,Z 213.96,A -85,B 0,C 180,E1 -9467.755,E2 -9467.755} C_VEL
LIN {X 0,Y 433.391,Z 188.851,A -85,B 0,C 180,E1 -9468.36,E2 -9468.36} C_VEL
LIN {X 0,Y 434.146,Z 173.694,A -85,B 0,C 180,E1 -9471.111,E2 -9471.111} C_VEL
LIN {X 0,Y 435.258,Z 156.212,A -85,B 0,C 180,E1 -9474.314,E2 -9474.314} C_VEL
LIN {X 0,Y 434.831,Z 151.819,A -85,B 0,C 180,E1 -9475.161,E2 -9475.161} C_VEL
LIN {X 0,Y 432.462,Z 139.617,A -85,B 0,C 180,E1 -9477.656,E2 -9477.656} C_VEL
LIN {X 0,Y 432.322,Z 139.63,A -85,B 0,C 180,E1 -9481.345,E2 -9481.345} C_VEL
LIN {X 0,Y 432.34,Z 139.627,A -85,B 0,C 180,E1 -9484.676,E2 -9484.676} C_VEL
LIN {X 0,Y 432.34,Z 139.631,A -85,B 0,C 180,E1 -9488.149,E2 -9488.149} C_VEL
LIN {X 0,Y 432.333,Z 139.632,A -85,B 0,C 180,E1 -9491.601,E2 -9491.601} C_VEL
LIN {X 0,Y 432.333,Z 139.629,A -85,B 0,C 180,E1 -9494.347,E2 -9494.347} C_VEL
LIN {X 0,Y 432.32,Z 139.63,A -85,B 0,C 180,E1 -9497.015,E2 -9497.015} C_VEL
LIN {X 0,Y 432.333,Z 139.633,A -85,B 0,C 180,E1 -9499.82,E2 -9499.82} C_VEL
LIN {X 0,Y 432.305,Z 139.632,A -85,B 0,C 180,E1 -9503.021,E2 -9503.021} C_VEL
LIN {X 0,Y 432.357,Z 139.627,A -85,B 0,C 180,E1 -9505.996,E2 -9505.996} C_VEL
LIN {X 0,Y 432.346,Z 139.633,A -85,B 0,C 180,E1 -9509.489,E2 -9509.489} C_VEL
LIN {X 0,Y 432.39,Z 139.623,A -85,B 0,C 180,E1 -9512.928,E2 -9512.928} C_VEL
LIN {X 0,Y 432.37,Z 139.624,A -85,B 0,C 180,E1 -9516.023,E2 -9516.023} C_VEL
LIN {X 0,Y 432.349,Z 139.63,A -85,B 0,C 180,E1 -9519.046,E2 -9519.046} C_VEL
LIN {X 0,Y 432.36,Z 139.624,A -85,B 0,C 180,E1 -9522.01,E2 -9522.01} C_VEL
LIN {X 0,Y 432.394,Z 139.625,A -85,B 0,C 180,E1 -9524.926,E2 -9524.926} C_VEL
LIN {X 0,Y 432.458,Z 139.613,A -85,B 0,C 180,E1 -9527.803,E2 -9527.803} C_VEL
LIN {X 0,Y 432.49,Z 139.609,A -85,B 0,C 180,E1 -9531.59,E2 -9531.59} C_VEL
LIN {X 0,Y 432.592,Z 139.597,A -85,B 0,C 180,E1 -9534.406,E2 -9534.406} C_VEL
LIN {X 0,Y 432.605,Z 139.594,A -85,B 0,C 180,E1 -9538.138,E2 -9538.138} C_VEL
LIN {X 0,Y 432.732,Z 139.578,A -85,B 0,C 180,E1 -9539.999,E2 -9539.999} C_VEL
LIN {X 0,Y 432.602,Z 139.602,A -85,B 0,C 180,E1 -9542.793,E2 -9542.793} C_VEL
LIN {X 0,Y 432.563,Z 139.604,A -85,B 0,C 180,E1 -9546.53,E2 -9546.53} C_VEL
LIN {X 0,Y 432.441,Z 139.615,A -85,B 0,C 180,E1 -9549.353,E2 -9549.353} C_VEL
LIN {X 0,Y 432.428,Z 139.62,A -85,B 0,C 180,E1 -9552.803,E2 -9552.803} C_VEL
LIN {X 0,Y 432.409,Z 139.625,A -85,B 0,C 180,E1 -9556.479,E2 -9556.479} C_VEL
LIN {X 0,Y 432.336,Z 139.629,A -85,B 0,C 180,E1 -9559.96,E2 -9559.96} C_VEL
LIN {X 0,Y 432.315,Z 139.631,A -85,B 0,C 180,E1 -9562.964,E2 -9562.964} C_VEL
LIN {X 0,Y 432.36,Z 139.628,A -85,B 0,C 180,E1 -9566.032,E2 -9566.032} C_VEL
LIN {X 0,Y 432.339,Z 139.627,A -85,B 0,C 180,E1 -9569.187,E2 -9569.187} C_VEL
LIN {X 0,Y 432.319,Z 139.634,A -85,B 0,C 180,E1 -9572.443,E2 -9572.443} C_VEL
LIN {X 0,Y 432.341,Z 139.629,A -85,B 0,C 180,E1 -9575.632,E2 -9575.632} C_VEL
LIN {X 0,Y 432.356,Z 139.625,A -85,B 0,C 180,E1 -9578.718,E2 -9578.718} C_VEL
LIN {X 0,Y 432.369,Z 139.628,A -85,B 0,C 180,E1 -9581.792,E2 -9581.792} C_VEL
LIN {X 0,Y 432.373,Z 139.625,A -85,B 0,C 180,E1 -9584.341,E2 -9584.341} C_VEL
LIN {X 0,Y 432.361,Z 139.624,A -85,B 0,C 180,E1 -9587.009,E2 -9587.009} C_VEL
LIN {X 0,Y 432.354,Z 139.633,A -85,B 0,C 180,E1 -9589.817,E2 -9589.817} C_VEL
LIN {X 0,Y 432.312,Z 139.631,A -85,B 0,C 180,E1 -9593.023,E2 -9593.023} C_VEL
LIN {X 0,Y 432.354,Z 139.629,A -85,B 0,C 180,E1 -9595.996,E2 -9595.996} C_VEL
LIN {X 0,Y 432.342,Z 139.632,A -85,B 0,C 180,E1 -9599.49,E2 -9599.49} C_VEL
LIN {X 0,Y 432.388,Z 139.622,A -85,B 0,C 180,E1 -9602.929,E2 -9602.929} C_VEL
LIN {X 0,Y 432.367,Z 139.625,A -85,B 0,C 180,E1 -9606.024,E2 -9606.024} C_VEL
LIN {X 0,Y 432.346,Z 139.629,A -85,B 0,C 180,E1 -9609.046,E2 -9609.046} C_VEL
LIN {X 0,Y 432.374,Z 139.623,A -85,B 0,C 180,E1 -9612.012,E2 -9612.012} C_VEL
LIN {X 0,Y 432.392,Z 139.623,A -85,B 0,C 180,E1 -9614.927,E2 -9614.927} C_VEL
LIN {X 0,Y 432.455,Z 139.614,A -85,B 0,C 180,E1 -9617.804,E2 -9617.804} C_VEL
LIN {X 0,Y 432.488,Z 139.611,A -85,B 0,C 180,E1 -9621.591,E2 -9621.591} C_VEL
LIN {X 0,Y 432.596,Z 139.595,A -85,B 0,C 180,E1 -9624.407,E2 -9624.407} C_VEL
LIN {X 0,Y 432.602,Z 139.594,A -85,B 0,C 180,E1 -9628.139,E2 -9628.139} C_VEL
LIN {X 0,Y 432.73,Z 139.578,A -85,B 0,C 180,E1 -9630.001,E2 -9630.001} C_VEL
LIN {X 0,Y 432.602,Z 139.6,A -85,B 0,C 180,E1 -9632.794,E2 -9632.794} C_VEL
LIN {X 0,Y 432.462,Z 139.613,A -85,B 0,C 180,E1 -9635.028,E2 -9635.028} C_VEL
LIN {X 0,Y 431.903,Z 139.682,A -85,B 0,C 180,E1 -9635.807,E2 -9635.807} C_VEL
LIN {X 0,Y 429.057,Z 140.04,A -85,B 0,C 180,E1 -9637.072,E2 -9637.072} C_VEL
LIN {X 0,Y 426.572,Z 140.348,A -85,B 0,C 180,E1 -9638.093,E2 -9638.093} C_VEL
LIN {X 0,Y 425.491,Z 140.487,A -85,B 0,C 180,E1 -9638.883,E2 -9638.883} C_VEL
LIN {X 0,Y 425.4,Z 140.491,A -85,B 0,C 180,E1 -9639.15,E2 -9639.15} C_VEL
LIN {X 0,Y 425.391,Z 140.498,A -85,B 0,C 180,E1 -9642.904,E2 -9642.904} C_VEL
LIN {X 0,Y 425.388,Z 140.505,A -85,B 0,C 180,E1 -9646.778,E2 -9646.778} C_VEL
LIN {X 0,Y 426.796,Z 148.745,A -85,B 0,C 180,E1 -9648.73,E2 -9648.73} C_VEL
LIN {X 0,Y 426.885,Z 152.148,A -85,B 0,C 180,E1 -9649.465,E2 -9649.465} C_VEL
LIN {X 0,Y 430.544,Z 170.361,A -85,B 0,C 180,E1 -9649.95,E2 -9649.95} C_VEL
LIN {X 0,Y 429.359,Z 259.5,A -85,B 0,C 180,E1 -9651.516,E2 -9651.516} C_VEL
LIN {X 0,Y 428.98,Z 272.937,A -85,B 0,C 180,E1 -9651.947,E2 -9651.947} C_VEL
LIN {X 0,Y 428.619,Z 285.332,A -85,B 0,C 180,E1 -9652.537,E2 -9652.537} C_VEL
LIN {X 0,Y 428.186,Z 295.803,A -85,B 0,C 180,E1 -9653.199,E2 -9653.199} C_VEL
LIN {X 0,Y 427.475,Z 307.476,A -85,B 0,C 180,E1 -9654.14,E2 -9654.14} C_VEL
LIN {X 0,Y 426.829,Z 318.216,A -85,B 0,C 180,E1 -9655.232,E2 -9655.232} C_VEL
LIN {X 0,Y 426.237,Z 327.757,A -85,B 0,C 180,E1 -9656.436,E2 -9656.436} C_VEL
LIN {X 0,Y 425.657,Z 336.48,A -85,B 0,C 180,E1 -9657.804,E2 -9657.804} C_VEL
LIN {X 0,Y 425.189,Z 343.952,A -85,B 0,C 180,E1 -9659.256,E2 -9659.256} C_VEL
LIN {X 0,Y 424.786,Z 350.446,A -85,B 0,C 180,E1 -9660.857,E2 -9660.857} C_VEL
LIN {X 0,Y 424.467,Z 355.21,A -85,B 0,C 180,E1 -9662.391,E2 -9662.391} C_VEL
LIN {X 0,Y 424.241,Z 359.023,A -85,B 0,C 180,E1 -9664.076,E2 -9664.076} C_VEL
LIN {X 0,Y 424.084,Z 361.424,A -85,B 0,C 180,E1 -9665.706,E2 -9665.706} C_VEL
LIN {X 0,Y 424.037,Z 362.605,A -85,B 0,C 180,E1 -9667.294,E2 -9667.294} C_VEL
LIN {X 0,Y 424.031,Z 362.6,A -85,B 0,C 180,E1 -9669.038,E2 -9669.038} C_VEL
LIN {X 0,Y 424.109,Z 361.739,A -85,B 0,C 180,E1 -9670.336,E2 -9670.336} C_VEL
LIN {X 0,Y 424.257,Z 359.839,A -85,B 0,C 180,E1 -9671.804,E2 -9671.804} C_VEL
LIN {X 0,Y 424.483,Z 356.998,A -85,B 0,C 180,E1 -9673.241,E2 -9673.241} C_VEL
LIN {X 0,Y 424.754,Z 352.253,A -85,B 0,C 180,E1 -9674.954,E2 -9674.954} C_VEL
LIN {X 0,Y 425.214,Z 345.867,A -85,B 0,C 180,E1 -9676.656,E2 -9676.656} C_VEL
LIN {X 0,Y 425.662,Z 339.537,A -85,B 0,C 180,E1 -9677.987,E2 -9677.987} C_VEL
LIN {X 0,Y 426.247,Z 331.696,A -85,B 0,C 180,E1 -9679.329,E2 -9679.329} C_VEL
LIN {X 0,Y 426.938,Z 321.775,A -85,B 0,C 180,E1 -9680.687,E2 -9680.687} C_VEL
LIN {X 0,Y 427.592,Z 311.322,A -85,B 0,C 180,E1 -9681.84,E2 -9681.84} C_VEL
LIN {X 0,Y 428.285,Z 301.329,A -85,B 0,C 180,E1 -9682.721,E2 -9682.721} C_VEL
LIN {X 0,Y 428.911,Z 290.056,A -85,B 0,C 180,E1 -9683.511,E2 -9683.511} C_VEL
LIN {X 0,Y 429.403,Z 277.656,A -85,B 0,C 180,E1 -9684.173,E2 -9684.173} C_VEL
LIN {X 0,Y 429.756,Z 264.703,A -85,B 0,C 180,E1 -9684.662,E2 -9684.662} C_VEL
LIN {X 0,Y 430.068,Z 249.447,A -85,B 0,C 180,E1 -9684.991,E2 -9684.991} C_VEL
LIN {X 0,Y 431.139,Z 170.588,A -85,B 0,C 180,E1 -9686.378,E2 -9686.378} C_VEL
LIN {X 0,Y 427.255,Z 152.747,A -85,B 0,C 180,E1 -9686.904,E2 -9686.904} C_VEL
LIN {X 0,Y 426.687,Z 147.063,A -85,B 0,C 180,E1 -9688.193,E2 -9688.193} C_VEL
LIN {X 0,Y 425.329,Z 140.506,A -85,B 0,C 180,E1 -9689.772,E2 -9689.772} C_VEL
LIN {X 0,Y 425.343,Z 140.507,A -85,B 0,C 180,E1 -9693.159,E2 -9693.159} C_VEL
LIN {X 0,Y 425.349,Z 140.505,A -85,B 0,C 180,E1 -9695.603,E2 -9695.603} C_VEL
LIN {X 0,Y 425.296,Z 140.512,A -85,B 0,C 180,E1 -9698.682,E2 -9698.682} C_VEL
LIN {X 0,Y 425.324,Z 140.503,A -85,B 0,C 180,E1 -9701.703,E2 -9701.703} C_VEL
LIN {X 0,Y 425.35,Z 140.503,A -85,B 0,C 180,E1 -9704.671,E2 -9704.671} C_VEL
LIN {X 0,Y 425.416,Z 140.494,A -85,B 0,C 180,E1 -9707.599,E2 -9707.599} C_VEL
LIN {X 0,Y 425.412,Z 140.494,A -85,B 0,C 180,E1 -9711.45,E2 -9711.45} C_VEL
LIN {X 0,Y 425.531,Z 140.484,A -85,B 0,C 180,E1 -9714.313,E2 -9714.313} C_VEL
LIN {X 0,Y 425.57,Z 140.477,A -85,B 0,C 180,E1 -9718.108,E2 -9718.108} C_VEL
LIN {X 0,Y 425.577,Z 140.47,A -85,B 0,C 180,E1 -9720.001,E2 -9720.001} C_VEL
LIN {X 0,Y 425.516,Z 140.473,A -85,B 0,C 180,E1 -9722.841,E2 -9722.841} C_VEL
LIN {X 0,Y 425.529,Z 140.48,A -85,B 0,C 180,E1 -9725.688,E2 -9725.688} C_VEL
LIN {X 0,Y 425.398,Z 140.493,A -85,B 0,C 180,E1 -9728.551,E2 -9728.551} C_VEL
LIN {X 0,Y 425.406,Z 140.492,A -85,B 0,C 180,E1 -9732.402,E2 -9732.402} C_VEL
LIN {X 0,Y 425.313,Z 140.503,A -85,B 0,C 180,E1 -9736.315,E2 -9736.315} C_VEL
LIN {X 0,Y 425.281,Z 140.506,A -85,B 0,C 180,E1 -9739.616,E2 -9739.616} C_VEL
LIN {X 0,Y 425.288,Z 140.506,A -85,B 0,C 180,E1 -9742.339,E2 -9742.339} C_VEL
LIN {X 0,Y 425.253,Z 140.516,A -85,B 0,C 180,E1 -9745.449,E2 -9745.449} C_VEL
LIN {X 0,Y 425.3,Z 140.505,A -85,B 0,C 180,E1 -9748.857,E2 -9748.857} C_VEL
LIN {X 0,Y 425.257,Z 140.508,A -85,B 0,C 180,E1 -9751.928,E2 -9751.928} C_VEL
LIN {X 0,Y 425.3,Z 140.506,A -85,B 0,C 180,E1 -9755.336,E2 -9755.336} C_VEL
LIN {X 0,Y 425.285,Z 140.509,A -85,B 0,C 180,E1 -9758.901,E2 -9758.901} C_VEL
LIN {X 0,Y 425.261,Z 140.517,A -85,B 0,C 180,E1 -9762.655,E2 -9762.655} C_VEL
LIN {X 0,Y 425.29,Z 140.51,A -85,B 0,C 180,E1 -9765.283,E2 -9765.283} C_VEL
LIN {X 0,Y 425.258,Z 140.516,A -85,B 0,C 180,E1 -9768.619,E2 -9768.619} C_VEL
LIN {X 0,Y 425.285,Z 140.509,A -85,B 0,C 180,E1 -9771.099,E2 -9771.099} C_VEL
LIN {X 0,Y 425.304,Z 140.509,A -85,B 0,C 180,E1 -9774.664,E2 -9774.664} C_VEL
LIN {X 0,Y 425.27,Z 140.519,A -85,B 0,C 180,E1 -9778.073,E2 -9778.073} C_VEL
LIN {X 0,Y 425.319,Z 140.507,A -85,B 0,C 180,E1 -9781.366,E2 -9781.366} C_VEL
LIN {X 0,Y 425.343,Z 140.631,A -85,B 0,C 180,E1 -9782.107,E2 -9782.107} C_VEL
LIN {X 0,Y 427.996,Z 153.245,A -85,B 0,C 180,E1 -9784.726,E2 -9784.726} C_VEL
LIN {X 0,Y 428.343,Z 157.323,A -85,B 0,C 180,E1 -9785.525,E2 -9785.525} C_VEL
LIN {X 0,Y 427.205,Z 174.934,A -85,B 0,C 180,E1 -9788.781,E2 -9788.781} C_VEL
LIN {X 0,Y 426.586,Z 187.512,A -85,B 0,C 180,E1 -9791.087,E2 -9791.087} C_VEL
LIN {X 0,Y 430.55,Z 213.867,A -85,B 0,C 180,E1 -9791.771,E2 -9791.771} C_VEL
LIN {X 0,Y 429.644,Z 296.557,A -85,B 0,C 180,E1 -9793.243,E2 -9793.243} C_VEL
LIN {X 0,Y 429.071,Z 310.433,A -85,B 0,C 180,E1 -9793.679,E2 -9793.679} C_VEL
LIN {X 0,Y 428.402,Z 323.469,A -85,B 0,C 180,E1 -9794.294,E2 -9794.294} C_VEL
LIN {X 0,Y 427.648,Z 336.112,A -85,B 0,C 180,E1 -9795.12,E2 -9795.12} C_VEL
LIN {X 0,Y 426.971,Z 347.024,A -85,B 0,C 180,E1 -9796.034,E2 -9796.034} C_VEL
LIN {X 0,Y 426.16,Z 357.597,A -85,B 0,C 180,E1 -9797.136,E2 -9797.136} C_VEL
LIN {X 0,Y 425.657,Z 366.81,A -85,B 0,C 180,E1 -9798.33,E2 -9798.33} C_VEL
LIN {X 0,Y 424.976,Z 375.801,A -85,B 0,C 180,E1 -9799.759,E2 -9799.759} C_VEL
LIN {X 0,Y 424.6,Z 383.043,A -85,B 0,C 180,E1 -9801.192,E2 -9801.192} C_VEL
LIN {X 0,Y 424.366,Z 387.944,A -85,B 0,C 180,E1 -9802.386,E2 -9802.386} C_VEL
LIN {X 0,Y 424.222,Z 392.433,A -85,B 0,C 180,E1 -9803.727,E2 -9803.727} C_VEL
LIN {X 0,Y 424.197,Z 396.353,A -85,B 0,C 180,E1 -9805.248,E2 -9805.248} C_VEL
LIN {X 0,Y 424.109,Z 398.22,A -85,B 0,C 180,E1 -9806.199,E2 -9806.199} C_VEL
LIN {X 0,Y 424.179,Z 399.63,A -85,B 0,C 180,E1 -9807.15,E2 -9807.15} C_VEL
LIN {X 0,Y 424.167,Z 400.637,A -85,B 0,C 180,E1 -9808.1,E2 -9808.1} C_VEL
LIN {X 0,Y 424.141,Z 401.249,A -85,B 0,C 180,E1 -9809.05,E2 -9809.05} C_VEL
LIN {X 0,Y 424.143,Z 401.44,A -85,B 0,C 180,E1 -9809.999,E2 -9809.999} C_VEL
LIN {X 0,Y 424.141,Z 401.205,A -85,B 0,C 180,E1 -9810.949,E2 -9810.949} C_VEL
LIN {X 0,Y 424.167,Z 400.578,A -85,B 0,C 180,E1 -9811.898,E2 -9811.898} C_VEL
LIN {X 0,Y 424.18,Z 399.554,A -85,B 0,C 180,E1 -9812.849,E2 -9812.849} C_VEL
LIN {X 0,Y 424.111,Z 398.087,A -85,B 0,C 180,E1 -9813.8,E2 -9813.8} C_VEL
LIN {X 0,Y 424.195,Z 395.07,A -85,B 0,C 180,E1 -9815.228,E2 -9815.228} C_VEL
LIN {X 0,Y 424.257,Z 390.976,A -85,B 0,C 180,E1 -9816.658,E2 -9816.658} C_VEL
LIN {X 0,Y 424.504,Z 384.68,A -85,B 0,C 180,E1 -9818.329,E2 -9818.329} C_VEL
LIN {X 0,Y 424.838,Z 377.817,A -85,B 0,C 180,E1 -9819.762,E2 -9819.762} C_VEL
LIN {X 0,Y 425.229,Z 370.813,A -85,B 0,C 180,E1 -9820.956,E2 -9820.956} C_VEL
LIN {X 0,Y 425.816,Z 362.383,A -85,B 0,C 180,E1 -9822.147,E2 -9822.147} C_VEL
LIN {X 0,Y 426.418,Z 351.987,A -85,B 0,C 180,E1 -9823.34,E2 -9823.34} C_VEL
LIN {X 0,Y 427.136,Z 340.261,A -85,B 0,C 180,E1 -9824.41,E2 -9824.41} C_VEL
LIN {X 0,Y 427.837,Z 328.637,A -85,B 0,C 180,E1 -9825.237,E2 -9825.237} C_VEL
LIN {X 0,Y 428.485,Z 316.59,A -85,B 0,C 180,E1 -9825.884,E2 -9825.884} C_VEL
LIN {X 0,Y 429.011,Z 303.585,A -85,B 0,C 180,E1 -9826.384,E2 -9826.384} C_VEL
LIN {X 0,Y 429.327,Z 289.699,A -85,B 0,C 180,E1 -9826.707,E2 -9826.707} C_VEL
LIN {X 0,Y 430.158,Z 214.545,A -85,B 0,C 180,E1 -9828.01,E2 -9828.01} C_VEL
LIN {X 0,Y 426.432,Z 188.657,A -85,B 0,C 180,E1 -9828.633,E2 -9828.633} C_VEL
LIN {X 0,Y 427.162,Z 174.628,A -85,B 0,C 180,E1 -9831.22,E2 -9831.22} C_VEL
LIN {X 0,Y 428.317,Z 157.146,A -85,B 0,C 180,E1 -9834.475,E2 -9834.475} C_VEL
LIN {X 0,Y 427.644,Z 151.698,A -85,B 0,C 180,E1 -9835.555,E2 -9835.555} C_VEL
LIN {X 0,Y 425.414,Z 140.497,A -85,B 0,C 180,E1 -9837.887,E2 -9837.887} C_VEL
LIN {X 0,Y 425.289,Z 140.506,A -85,B 0,C 180,E1 -9840.815,E2 -9840.815} C_VEL
LIN {X 0,Y 425.312,Z 140.506,A -85,B 0,C 180,E1 -9844.287,E2 -9844.287} C_VEL
LIN {X 0,Y 425.28,Z 140.511,A -85,B 0,C 180,E1 -9847.693,E2 -9847.693} C_VEL
LIN {X 0,Y 425.284,Z 140.506,A -85,B 0,C 180,E1 -9850.52,E2 -9850.52} C_VEL
LIN {X 0,Y 425.257,Z 140.511,A -85,B 0,C 180,E1 -9853.35,E2 -9853.35} C_VEL
LIN {X 0,Y 425.257,Z 140.509,A -85,B 0,C 180,E1 -9856.649,E2 -9856.649} C_VEL
LIN {X 0,Y 425.285,Z 140.51,A -85,B 0,C 180,E1 -9859.872,E2 -9859.872} C_VEL
LIN {X 0,Y 425.277,Z 140.507,A -85,B 0,C 180,E1 -9862.488,E2 -9862.488} C_VEL
LIN {X 0,Y 425.305,Z 140.507,A -85,B 0,C 180,E1 -9865.817,E2 -9865.817} C_VEL
LIN {X 0,Y 425.289,Z 140.509,A -85,B 0,C 180,E1 -9869.238,E2 -9869.238} C_VEL
LIN {X 0,Y 425.348,Z 140.498,A -85,B 0,C 180,E1 -9872.442,E2 -9872.442} C_VEL
LIN {X 0,Y 425.35,Z 140.502,A -85,B 0,C 180,E1 -9875.602,E2 -9875.602} C_VEL
LIN {X 0,Y 425.292,Z 140.506,A -85,B 0,C 180,E1 -9878.681,E2 -9878.681} C_VEL
LIN {X 0,Y 425.32,Z 140.503,A -85,B 0,C 180,E1 -9881.702,E2 -9881.702} C_VEL
LIN {X 0,Y 425.347,Z 140.5,A -85,B 0,C 180,E1 -9884.67,E2 -9884.67} C_VEL
LIN {X 0,Y 425.411,Z 140.492,A -85,B 0,C 180,E1 -9887.598,E2 -9887.598} C_VEL
LIN {X 0,Y 425.441,Z 140.489,A -85,B 0,C 180,E1 -9891.449,E2 -9891.449} C_VEL
LIN {X 0,Y 425.549,Z 140.474,A -85,B 0,C 180,E1 -9894.313,E2 -9894.313} C_VEL
LIN {X 0,Y 425.574,Z 140.47,A -85,B 0,C 180,E1 -9898.107,E2 -9898.107} C_VEL
LIN {X 0,Y 425.701,Z 140.454,A -85,B 0,C 180,E1 -9899.999,E2 -9899.999} C_VEL
LIN {X 0,Y 425.554,Z 140.479,A -85,B 0,C 180,E1 -9902.839,E2 -9902.839} C_VEL
LIN {X 0,Y 425.521,Z 140.483,A -85,B 0,C 180,E1 -9906.638,E2 -9906.638} C_VEL
LIN {X 0,Y 425.399,Z 140.491,A -85,B 0,C 180,E1 -9909.509,E2 -9909.509} C_VEL
LIN {X 0,Y 425.39,Z 140.496,A -85,B 0,C 180,E1 -9912.903,E2 -9912.903} C_VEL
LIN {X 0,Y 425.358,Z 140.503,A -85,B 0,C 180,E1 -9916.605,E2 -9916.605} C_VEL
LIN {X 0,Y 425.325,Z 140.501,A -85,B 0,C 180,E1 -9919.635,E2 -9919.635} C_VEL
LIN {X 0,Y 425.303,Z 140.503,A -85,B 0,C 180,E1 -9923.365,E2 -9923.365} C_VEL
LIN {X 0,Y 425.345,Z 140.5,A -85,B 0,C 180,E1 -9926.844,E2 -9926.844} C_VEL
LIN {X 0,Y 425.287,Z 140.507,A -85,B 0,C 180,E1 -9929.719,E2 -9929.719} C_VEL
LIN {X 0,Y 425.277,Z 140.507,A -85,B 0,C 180,E1 -9933.048,E2 -9933.048} C_VEL
LIN {X 0,Y 425.28,Z 140.511,A -85,B 0,C 180,E1 -9935.929,E2 -9935.929} C_VEL
LIN {X 0,Y 425.309,Z 140.503,A -85,B 0,C 180,E1 -9939.046,E2 -9939.046} C_VEL
LIN {X 0,Y 425.327,Z 140.501,A -85,B 0,C 180,E1 -9942.646,E2 -9942.646} C_VEL
LIN {X 0,Y 425.329,Z 140.506,A -85,B 0,C 180,E1 -9946.054,E2 -9946.054} C_VEL
LIN {X 0,Y 425.305,Z 140.503,A -85,B 0,C 180,E1 -9948.626,E2 -9948.626} C_VEL
LIN {X 0,Y 425.32,Z 140.502,A -85,B 0,C 180,E1 -9951.104,E2 -9951.104} C_VEL
LIN {X 0,Y 425.295,Z 140.504,A -85,B 0,C 180,E1 -9954.664,E2 -9954.664} C_VEL
LIN {X 0,Y 425.26,Z 140.511,A -85,B 0,C 180,E1 -9958.073,E2 -9958.073} C_VEL
LIN {X 0,Y 425.326,Z 140.505,A -85,B 0,C 180,E1 -9961.368,E2 -9961.368} C_VEL
LIN {X 0,Y 425.29,Z 140.505,A -85,B 0,C 180,E1 -9964.555,E2 -9964.555} C_VEL
LIN {X 0,Y 425.283,Z 140.511,A -85,B 0,C 180,E1 -9967.662,E2 -9967.662} C_VEL
LIN {X 0,Y 425.357,Z 140.497,A -85,B 0,C 180,E1 -9970.704,E2 -9970.704} C_VEL
LIN {X 0,Y 425.384,Z 140.496,A -85,B 0,C 180,E1 -9973.689,E2 -9973.689} C_VEL
LIN {X 0,Y 425.408,Z 140.493,A -85,B 0,C 180,E1 -9977.599,E2 -9977.599} C_VEL
LIN {X 0,Y 425.438,Z 140.49,A -85,B 0,C 180,E1 -9981.45,E2 -9981.45} C_VEL
LIN {X 0,Y 425.552,Z 140.473,A -85,B 0,C 180,E1 -9984.314,E2 -9984.314} C_VEL
LIN {X 0,Y 425.572,Z 140.47,A -85,B 0,C 180,E1 -9988.108,E2 -9988.108} C_VEL
LIN {X 0,Y 425.7,Z 140.454,A -85,B 0,C 180,E1 -9990.001,E2 -9990.001} C_VEL
LIN {X 0,Y 425.554,Z 140.478,A -85,B 0,C 180,E1 -9992.84,E2 -9992.84} C_VEL
LIN {X 0,Y 425.529,Z 140.48,A -85,B 0,C 180,E1 -9996.639,E2 -9996.639} C_VEL
LIN {X 0,Y 425.4,Z 140.491,A -85,B 0,C 180,E1 -9999.15,E2 -9999.15} C_VEL
LIN {X 0,Y 424.728,Z 140.576,A -85,B 0,C 180,E1 -9999.94,E2 -9999.94} C_VEL
LIN {X 0,Y 421.88,Z 140.934,A -85,B 0,C 180,E1 -10001.224,E2 -10001.224} C_VEL
LIN {X 0,Y 419.464,Z 141.236,A -85,B 0,C 180,E1 -10002.26,E2 -10002.26} C_VEL
LIN {X 0,Y 418.413,Z 141.367,A -85,B 0,C 180,E1 -10003.061,E2 -10003.061} C_VEL
LIN {X 0,Y 418.32,Z 141.377,A -85,B 0,C 180,E1 -10003.332,E2 -10003.332} C_VEL
LIN {X 0,Y 418.384,Z 141.454,A -85,B 0,C 180,E1 -10006.593,E2 -10006.593} C_VEL
LIN {X 0,Y 419.877,Z 150.66,A -85,B 0,C 180,E1 -10008.797,E2 -10008.797} C_VEL
LIN {X 0,Y 419.982,Z 152.506,A -85,B 0,C 180,E1 -10009.173,E2 -10009.173} C_VEL
LIN {X 0,Y 423.773,Z 171.404,A -85,B 0,C 180,E1 -10009.687,E2 -10009.687} C_VEL
LIN {X 0,Y 422.515,Z 259.737,A -85,B 0,C 180,E1 -10011.264,E2 -10011.264} C_VEL
LIN {X 0,Y 422.135,Z 273.406,A -85,B 0,C 180,E1 -10011.711,E2 -10011.711} C_VEL
LIN {X 0,Y 421.7,Z 286.379,A -85,B 0,C 180,E1 -10012.346,E2 -10012.346} C_VEL
LIN {X 0,Y 421.192,Z 298.273,A -85,B 0,C 180,E1 -10013.14,E2 -10013.14} C_VEL
LIN {X 0,Y 420.5,Z 308.949,A -85,B 0,C 180,E1 -10014.042,E2 -10014.042} C_VEL
LIN {X 0,Y 419.851,Z 319.096,A -85,B 0,C 180,E1 -10015.106,E2 -10015.106} C_VEL
LIN {X 0,Y 419.208,Z 328.827,A -85,B 0,C 180,E1 -10016.377,E2 -10016.377} C_VEL
LIN {X 0,Y 418.599,Z 337.704,A -85,B 0,C 180,E1 -10017.817,E2 -10017.817} C_VEL
LIN {X 0,Y 418.159,Z 344.452,A -85,B 0,C 180,E1 -10019.171,E2 -10019.171} C_VEL
LIN {X 0,Y 417.751,Z 350.218,A -85,B 0,C 180,E1 -10020.601,E2 -10020.601} C_VEL
LIN {X 0,Y 417.479,Z 354.75,A -85,B 0,C 180,E1 -10022.025,E2 -10022.025} C_VEL
LIN {X 0,Y 417.191,Z 358.865,A -85,B 0,C 180,E1 -10023.775,E2 -10023.775} C_VEL
LIN {X 0,Y 417.059,Z 360.848,A -85,B 0,C 180,E1 -10024.957,E2 -10024.957} C_VEL
LIN {X 0,Y 416.962,Z 362.189,A -85,B 0,C 180,E1 -10026.153,E2 -10026.153} C_VEL
LIN {X 0,Y 416.935,Z 363.009,A -85,B 0,C 180,E1 -10027.605,E2 -10027.605} C_VEL
LIN {X 0,Y 416.965,Z 362.882,A -85,B 0,C 180,E1 -10029.166,E2 -10029.166} C_VEL
LIN {X 0,Y 417.092,Z 361.304,A -85,B 0,C 180,E1 -10031.084,E2 -10031.084} C_VEL
LIN {X 0,Y 417.255,Z 359.345,A -85,B 0,C 180,E1 -10032.357,E2 -10032.357} C_VEL
LIN {X 0,Y 417.447,Z 356.608,A -85,B 0,C 180,E1 -10033.652,E2 -10033.652} C_VEL
LIN {X 0,Y 417.72,Z 352.745,A -85,B 0,C 180,E1 -10035.039,E2 -10035.039} C_VEL
LIN {X 0,Y 418.177,Z 346.789,A -85,B 0,C 180,E1 -10036.675,E2 -10036.675} C_VEL
LIN {X 0,Y 418.725,Z 339.49,A -85,B 0,C 180,E1 -10038.246,E2 -10038.246} C_VEL
LIN {X 0,Y 419.386,Z 331.229,A -85,B 0,C 180,E1 -10039.654,E2 -10039.654} C_VEL
LIN {X 0,Y 420.086,Z 321.489,A -85,B 0,C 180,E1 -10040.991,E2 -10040.991} C_VEL
LIN {X 0,Y 420.786,Z 311.133,A -85,B 0,C 180,E1 -10042.136,E2 -10042.136} C_VEL
LIN {X 0,Y 421.644,Z 299.581,A -85,B 0,C 180,E1 -10043.138,E2 -10043.138} C_VEL
LIN {X 0,Y 422.278,Z 287.92,A -85,B 0,C 180,E1 -10043.933,E2 -10043.933} C_VEL
LIN {X 0,Y 422.715,Z 274.968,A -85,B 0,C 180,E1 -10044.593,E2 -10044.593} C_VEL
LIN {X 0,Y 423.113,Z 261.283,A -85,B 0,C 180,E1 -10045.056,E2 -10045.056} C_VEL
LIN {X 0,Y 423.996,Z 204.354,A -85,B 0,C 180,E1 -10046.099,E2 -10046.099} C_VEL
LIN {X 0,Y 424.423,Z 171.152,A -85,B 0,C 180,E1 -10046.7,E2 -10046.7} C_VEL
LIN {X 0,Y 420.355,Z 153.016,A -85,B 0,C 180,E1 -10047.27,E2 -10047.27} C_VEL
LIN {X 0,Y 419.249,Z 145.976,A -85,B 0,C 180,E1 -10048.921,E2 -10048.921} C_VEL
LIN {X 0,Y 418.28,Z 141.383,A -85,B 0,C 180,E1 -10050.079,E2 -10050.079} C_VEL
LIN {X 0,Y 418.307,Z 141.383,A -85,B 0,C 180,E1 -10053.024,E2 -10053.024} C_VEL
LIN {X 0,Y 418.276,Z 141.384,A -85,B 0,C 180,E1 -10056.219,E2 -10056.219} C_VEL
LIN {X 0,Y 418.253,Z 141.388,A -85,B 0,C 180,E1 -10059.338,E2 -10059.338} C_VEL
LIN {X 0,Y 418.283,Z 141.382,A -85,B 0,C 180,E1 -10062.397,E2 -10062.397} C_VEL
LIN {X 0,Y 418.305,Z 141.381,A -85,B 0,C 180,E1 -10065.404,E2 -10065.404} C_VEL
LIN {X 0,Y 418.318,Z 141.382,A -85,B 0,C 180,E1 -10068.37,E2 -10068.37} C_VEL
LIN {X 0,Y 418.382,Z 141.371,A -85,B 0,C 180,E1 -10071.305,E2 -10071.305} C_VEL
LIN {X 0,Y 418.489,Z 141.36,A -85,B 0,C 180,E1 -10074.217,E2 -10074.217} C_VEL
LIN {X 0,Y 418.539,Z 141.353,A -85,B 0,C 180,E1 -10078.076,E2 -10078.076} C_VEL
LIN {X 0,Y 418.415,Z 141.364,A -85,B 0,C 180,E1 -10080.963,E2 -10080.963} C_VEL
LIN {X 0,Y 418.473,Z 141.351,A -85,B 0,C 180,E1 -10082.888,E2 -10082.888} C_VEL
LIN {X 0,Y 418.487,Z 141.358,A -85,B 0,C 180,E1 -10085.784,E2 -10085.784} C_VEL
LIN {X 0,Y 418.371,Z 141.368,A -85,B 0,C 180,E1 -10088.696,E2 -10088.696} C_VEL
LIN {X 0,Y 418.302,Z 141.373,A -85,B 0,C 180,E1 -10091.632,E2 -10091.632} C_VEL
LIN {X 0,Y 418.281,Z 141.384,A -85,B 0,C 180,E1 -10093.606,E2 -10093.606} C_VEL
LIN {X 0,Y 418.255,Z 141.381,A -85,B 0,C 180,E1 -10096.707,E2 -10096.707} C_VEL
LIN {X 0,Y 418.228,Z 141.385,A -85,B 0,C 180,E1 -10099.772,E2 -10099.772} C_VEL
LIN {X 0,Y 418.227,Z 141.386,A -85,B 0,C 180,E1 -10102.737,E2 -10102.737} C_VEL
LIN {X 0,Y 418.214,Z 141.389,A -85,B 0,C 180,E1 -10105.908,E2 -10105.908} C_VEL
LIN {X 0,Y 418.259,Z 141.386,A -85,B 0,C 180,E1 -10109.163,E2 -10109.163} C_VEL
LIN {X 0,Y 418.253,Z 141.385,A -85,B 0,C 180,E1 -10112.842,E2 -10112.842} C_VEL
LIN {X 0,Y 418.249,Z 141.383,A -85,B 0,C 180,E1 -10116.237,E2 -10116.237} C_VEL
LIN {X 0,Y 418.205,Z 141.39,A -85,B 0,C 180,E1 -10119.688,E2 -10119.688} C_VEL
LIN {X 0,Y 418.212,Z 141.391,A -85,B 0,C 180,E1 -10122.318,E2 -10122.318} C_VEL
LIN {X 0,Y 418.241,Z 141.389,A -85,B 0,C 180,E1 -10125.108,E2 -10125.108} C_VEL
LIN {X 0,Y 418.228,Z 141.39,A -85,B 0,C 180,E1 -10127.765,E2 -10127.765} C_VEL
LIN {X 0,Y 418.243,Z 141.387,A -85,B 0,C 180,E1 -10131.556,E2 -10131.556} C_VEL
LIN {X 0,Y 418.264,Z 141.383,A -85,B 0,C 180,E1 -10135.159,E2 -10135.159} C_VEL
LIN {X 0,Y 418.251,Z 141.391,A -85,B 0,C 180,E1 -10137.472,E2 -10137.472} C_VEL
LIN {X 0,Y 418.269,Z 141.384,A -85,B 0,C 180,E1 -10140.896,E2 -10140.896} C_VEL
LIN {X 0,Y 418.291,Z 141.475,A -85,B 0,C 180,E1 -10141.8,E2 -10141.8} C_VEL
LIN {X 0,Y 420.886,Z 153.653,A -85,B 0,C 180,E1 -10144.383,E2 -10144.383} C_VEL
LIN {X 0,Y 421.454,Z 158.501,A -85,B 0,C 180,E1 -10145.361,E2 -10145.361} C_VEL
LIN {X 0,Y 420.187,Z 177.432,A -85,B 0,C 180,E1 -10148.923,E2 -10148.923} C_VEL
LIN {X 0,Y 419.694,Z 187.417,A -85,B 0,C 180,E1 -10150.749,E2 -10150.749} C_VEL
LIN {X 0,Y 423.725,Z 213.499,A -85,B 0,C 180,E1 -10151.44,E2 -10151.44} C_VEL
LIN {X 0,Y 423.835,Z 222.007,A -85,B 0,C 180,E1 -10151.604,E2 -10151.604} C_VEL
LIN {X 0,Y 422.878,Z 296.812,A -85,B 0,C 180,E1 -10152.967,E2 -10152.967} C_VEL
LIN {X 0,Y 422.274,Z 310.463,A -85,B 0,C 180,E1 -10153.409,E2 -10153.409} C_VEL
LIN {X 0,Y 421.564,Z 323.374,A -85,B 0,C 180,E1 -10154.033,E2 -10154.033} C_VEL
LIN {X 0,Y 420.786,Z 335.964,A -85,B 0,C 180,E1 -10154.872,E2 -10154.872} C_VEL
LIN {X 0,Y 420.024,Z 347.214,A -85,B 0,C 180,E1 -10155.833,E2 -10155.833} C_VEL
LIN {X 0,Y 419.236,Z 357.38,A -85,B 0,C 180,E1 -10156.919,E2 -10156.919} C_VEL
LIN {X 0,Y 418.655,Z 366.574,A -85,B 0,C 180,E1 -10158.132,E2 -10158.132} C_VEL
LIN {X 0,Y 417.953,Z 375.554,A -85,B 0,C 180,E1 -10159.585,E2 -10159.585} C_VEL
LIN {X 0,Y 417.521,Z 382.777,A -85,B 0,C 180,E1 -10161.042,E2 -10161.042} C_VEL
LIN {X 0,Y 417.254,Z 389.373,A -85,B 0,C 180,E1 -10162.742,E2 -10162.742} C_VEL
LIN {X 0,Y 417.083,Z 393.738,A -85,B 0,C 180,E1 -10164.197,E2 -10164.197} C_VEL
LIN {X 0,Y 417.103,Z 396.061,A -85,B 0,C 180,E1 -10165.167,E2 -10165.167} C_VEL
LIN {X 0,Y 417.024,Z 397.916,A -85,B 0,C 180,E1 -10166.134,E2 -10166.134} C_VEL
LIN {X 0,Y 417.076,Z 399.322,A -85,B 0,C 180,E1 -10167.102,E2 -10167.102} C_VEL
LIN {X 0,Y 417.093,Z 400.325,A -85,B 0,C 180,E1 -10168.068,E2 -10168.068} C_VEL
LIN {X 0,Y 417.06,Z 400.932,A -85,B 0,C 180,E1 -10169.034,E2 -10169.034} C_VEL
LIN {X 0,Y 417.059,Z 401.113,A -85,B 0,C 180,E1 -10169.999,E2 -10169.999} C_VEL
LIN {X 0,Y 417.06,Z 400.872,A -85,B 0,C 180,E1 -10170.965,E2 -10170.965} C_VEL
LIN {X 0,Y 417.093,Z 400.24,A -85,B 0,C 180,E1 -10171.931,E2 -10171.931} C_VEL
LIN {X 0,Y 417.077,Z 399.209,A -85,B 0,C 180,E1 -10172.897,E2 -10172.897} C_VEL
LIN {X 0,Y 417.025,Z 397.73,A -85,B 0,C 180,E1 -10173.865,E2 -10173.865} C_VEL
LIN {X 0,Y 417.107,Z 394.698,A -85,B 0,C 180,E1 -10175.317,E2 -10175.317} C_VEL
LIN {X 0,Y 417.178,Z 390.586,A -85,B 0,C 180,E1 -10176.772,E2 -10176.772} C_VEL
LIN {X 0,Y 417.446,Z 384.268,A -85,B 0,C 180,E1 -10178.471,E2 -10178.471} C_VEL
LIN {X 0,Y 417.796,Z 377.38,A -85,B 0,C 180,E1 -10179.928,E2 -10179.928} C_VEL
LIN {X 0,Y 418.234,Z 370.348,A -85,B 0,C 180,E1 -10181.142,E2 -10181.142} C_VEL
LIN {X 0,Y 418.815,Z 361.88,A -85,B 0,C 180,E1 -10182.354,E2 -10182.354} C_VEL
LIN {X 0,Y 419.458,Z 351.418,A -85,B 0,C 180,E1 -10183.566,E2 -10183.566} C_VEL
LIN {X 0,Y 420.234,Z 339.639,A -85,B 0,C 180,E1 -10184.652,E2 -10184.652} C_VEL
LIN {X 0,Y 420.973,Z 327.897,A -85,B 0,C 180,E1 -10185.492,E2 -10185.492} C_VEL
LIN {X 0,Y 421.665,Z 315.724,A -85,B 0,C 180,E1 -10186.148,E2 -10186.148} C_VEL
LIN {X 0,Y 422.15,Z 303.408,A -85,B 0,C 180,E1 -10186.626,E2 -10186.626} C_VEL
LIN {X 0,Y 422.49,Z 289.664,A -85,B 0,C 180,E1 -10186.955,E2 -10186.955} C_VEL
LIN {X 0,Y 423.282,Z 214.611,A -85,B 0,C 180,E1 -10188.283,E2 -10188.283} C_VEL
LIN {X 0,Y 419.463,Z 188.289,A -85,B 0,C 180,E1 -10188.942,E2 -10188.942} C_VEL
LIN {X 0,Y 420.477,Z 171.519,A -85,B 0,C 180,E1 -10192.09,E2 -10192.09} C_VEL
LIN {X 0,Y 421.383,Z 158.07,A -85,B 0,C 180,E1 -10194.642,E2 -10194.642} C_VEL
LIN {X 0,Y 420.096,Z 149.857,A -85,B 0,C 180,E1 -10196.316,E2 -10196.316} C_VEL
LIN {X 0,Y 418.359,Z 141.374,A -85,B 0,C 180,E1 -10198.126,E2 -10198.126} C_VEL
LIN {X 0,Y 418.212,Z 141.388,A -85,B 0,C 180,E1 -10201.395,E2 -10201.395} C_VEL
LIN {X 0,Y 418.266,Z 141.381,A -85,B 0,C 180,E1 -10204.58,E2 -10204.58} C_VEL
LIN {X 0,Y 418.23,Z 141.391,A -85,B 0,C 180,E1 -10207.833,E2 -10207.833} C_VEL
LIN {X 0,Y 418.223,Z 141.385,A -85,B 0,C 180,E1 -10210.947,E2 -10210.947} C_VEL
LIN {X 0,Y 418.21,Z 141.394,A -85,B 0,C 180,E1 -10213.729,E2 -10213.729} C_VEL
LIN {X 0,Y 418.208,Z 141.388,A -85,B 0,C 180,E1 -10216.448,E2 -10216.448} C_VEL
LIN {X 0,Y 418.222,Z 141.387,A -85,B 0,C 180,E1 -10219.13,E2 -10219.13} C_VEL
LIN {X 0,Y 418.225,Z 141.386,A -85,B 0,C 180,E1 -10222.166,E2 -10222.166} C_VEL
LIN {X 0,Y 418.263,Z 141.386,A -85,B 0,C 180,E1 -10225.419,E2 -10225.419} C_VEL
